gfCNCPoint5[23995] = {X 332.1055, Y 45.0114, Z -7.1667, A 0.000, B 0.000, C 0.000 }
gfCNCPoint5[23996] = {X 330.6899, Y 43.7933, Z -7.1667, A 0.000, B 0.000, C 0.000 }
gfCNCPoint5[23997] = {X 329.7573, Y 43.7998, Z -7.1667, A 0.000, B 0.000, C 0.000 }
gfCNCPoint5[23998] = {X 328.8457, Y 43.6022, Z -7.1667, A 0.000, B 0.000, C 0.000 }
gfCNCPoint5[23999] = {X 327.9994, Y 43.2101, Z -7.1667, A 0.000, B 0.000, C 0.000 }
gfCNCPoint5[24000] = {X 327.2594, Y 42.6425, Z -7.1667, A 0.000, B 0.000, C 0.000 }
gfCNCPoint5[24001] = {X 326.6366, Y 42.0352, Z -7.1667, A 0.000, B 0.000, C 0.000 }
gfCNCPoint5[24002] = {X 326.0198, Y 41.2760, Z -7.1667, A 0.000, B 0.000, C 0.000 }
gfCNCPoint5[24003] = {X 325.5934, Y 40.3956, Z -7.1667, A 0.000, B 0.000, C 0.000 }
gfCNCPoint5[24004] = {X 325.3802, Y 39.4410, Z -7.1667, A 0.000, B 0.000, C 0.000 }
gfCNCPoint5[24005] = {X 325.3913, Y 38.4628, Z -7.1667, A 0.000, B 0.000, C 0.000 }
gfCNCPoint5[24006] = {X 325.6264, Y 37.5133, Z -7.1667, A 0.000, B 0.000, C 0.000 }
gfCNCPoint5[24007] = {X 326.0727, Y 36.6429, Z -7.1667, A 0.000, B 0.000, C 0.000 }
gfCNCPoint5[24008] = {X 330.3061, Y 30.3131, Z -7.1667, A 0.000, B 0.000, C 0.000 }
gfCNCPoint5[24009] = {X 330.8964, Y 29.6095, Z -7.1667, A 0.000, B 0.000, C 0.000 }
gfCNCPoint5[24010] = {X 331.6243, Y 29.0495, Z -7.1667, A 0.000, B 0.000, C 0.000 }
gfCNCPoint5[24011] = {X 332.4558, Y 28.6593, Z -7.1667, A 0.000, B 0.000, C 0.000 }
gfCNCPoint5[24012] = {X 333.3518, Y 28.4574, Z -7.1667, A 0.000, B 0.000, C 0.000 }
gfCNCPoint5[24013] = {X 334.2702, Y 28.4532, Z -7.1667, A 0.000, B 0.000, C 0.000 }
gfCNCPoint5[24014] = {X 335.1680, Y 28.6468, Z -7.1667, A 0.000, B 0.000, C 0.000 }
gfCNCPoint5[24015] = {X 336.0031, Y 29.0293, Z -7.1667, A 0.000, B 0.000, C 0.000 }
gfCNCPoint5[24016] = {X 336.7362, Y 29.5826, Z -7.1667, A 0.000, B 0.000, C 0.000 }
gfCNCPoint5[24017] = {X 337.3723, Y 30.1953, Z -7.1667, A 0.000, B 0.000, C 0.000 }
gfCNCPoint5[24018] = {X 338.0008, Y 30.9797, Z -7.1667, A 0.000, B 0.000, C 0.000 }
gfCNCPoint5[24019] = {X 338.4269, Y 31.8901, Z -7.1667, A 0.000, B 0.000, C 0.000 }
gfCNCPoint5[24020] = {X 338.6268, Y 32.8751, Z -7.1667, A 0.000, B 0.000, C 0.000 }
gfCNCPoint5[24021] = {X 338.5892, Y 33.8795, Z -7.1667, A 0.000, B 0.000, C 0.000 }
gfCNCPoint5[24022] = {X 339.4394, Y 34.6548, Z -7.1667, A 0.000, B 0.000, C 0.000 }
gfCNCPoint5[24023] = {X 340.5845, Y 35.5676, Z -7.1667, A 0.000, B 0.000, C 0.000 }
gfCNCPoint5[24024] = {X 341.8428, Y 36.3165, Z -7.1667, A 0.000, B 0.000, C 0.000 }
gfCNCPoint5[24025] = {X 343.1911, Y 36.8877, Z -7.1667, A 0.000, B 0.000, C 0.000 }
gfCNCPoint5[24026] = {X 344.6045, Y 37.2707, Z -7.1667, A 0.000, B 0.000, C 0.000 }
gfCNCPoint5[24027] = {X 346.0568, Y 37.4583, Z -7.1667, A 0.000, B 0.000, C 0.000 }
gfCNCPoint5[24028] = {X 347.5211, Y 37.4471, Z -7.1667, A 0.000, B 0.000, C 0.000 }
gfCNCPoint5[24029] = {X 348.6869, Y 37.3101, Z -7.1667, A 0.000, B 0.000, C 0.000 }
gfCNCPoint5[24030] = {X 349.8249, Y 37.0222, Z -7.1667, A 0.000, B 0.000, C 0.000 }
gfCNCPoint5[24031] = {X 350.9155, Y 36.5881, Z -7.1667, A 0.000, B 0.000, C 0.000 }
gfCNCPoint5[24032] = {X 351.9402, Y 36.0155, Z -7.1667, A 0.000, B 0.000, C 0.000 }
gfCNCPoint5[24033] = {X 352.8814, Y 35.3139, Z -7.1667, A 0.000, B 0.000, C 0.000 }
gfCNCPoint5[24034] = {X 354.0420, Y 34.1861, Z -7.1667, A 0.000, B 0.000, C 0.000 }
gfCNCPoint5[24035] = {X 355.0465, Y 32.9171, Z -7.1667, A 0.000, B 0.000, C 0.000 }
gfCNCPoint5[24036] = {X 355.8777, Y 31.5284, Z -7.1667, A 0.000, B 0.000, C 0.000 }
gfCNCPoint5[24037] = {X 356.5216, Y 30.0436, Z -7.1667, A 0.000, B 0.000, C 0.000 }
gfCNCPoint5[24038] = {X 356.9674, Y 28.4878, Z -7.1667, A 0.000, B 0.000, C 0.000 }
gfCNCPoint5[24039] = {X 357.2419, Y 26.7920, Z -7.1667, A 0.000, B 0.000, C 0.000 }
gfCNCPoint5[24040] = {X 357.3537, Y 25.0778, Z -7.1667, A 0.000, B 0.000, C 0.000 }
gfCNCPoint5[24041] = {X 357.3018, Y 23.3607, Z -7.1667, A 0.000, B 0.000, C 0.000 }
gfCNCPoint5[24042] = {X 357.0867, Y 21.6563, Z -7.1667, A 0.000, B 0.000, C 0.000 }
gfCNCPoint5[24043] = {X 356.7306, Y 20.1305, Z -7.1667, A 0.000, B 0.000, C 0.000 }
gfCNCPoint5[24044] = {X 356.1774, Y 18.6646, Z -7.1667, A 0.000, B 0.000, C 0.000 }
gfCNCPoint5[24045] = {X 355.4366, Y 17.2839, Z -7.1667, A 0.000, B 0.000, C 0.000 }
gfCNCPoint5[24046] = {X 354.5211, Y 16.0124, Z -7.1667, A 0.000, B 0.000, C 0.000 }
gfCNCPoint5[24047] = {X 353.6429, Y 15.0774, Z -7.1667, A 0.000, B 0.000, C 0.000 }
gfCNCPoint5[24048] = {X 352.6435, Y 14.2732, Z -7.1667, A 0.000, B 0.000, C 0.000 }
gfCNCPoint5[24049] = {X 351.5422, Y 13.6154, Z -7.1667, A 0.000, B 0.000, C 0.000 }
gfCNCPoint5[24050] = {X 350.3604, Y 13.1166, Z -7.1667, A 0.000, B 0.000, C 0.000 }
gfCNCPoint5[24051] = {X 349.1209, Y 12.7865, Z -7.1667, A 0.000, B 0.000, C 0.000 }
gfCNCPoint5[24052] = {X 347.3426, Y 12.5648, Z -7.1667, A 0.000, B 0.000, C 0.000 }
gfCNCPoint5[24053] = {X 345.5506, Y 12.5817, Z -7.1667, A 0.000, B 0.000, C 0.000 }
gfCNCPoint5[24054] = {X 343.7768, Y 12.8368, Z -7.1667, A 0.000, B 0.000, C 0.000 }
gfCNCPoint5[24055] = {X 342.0527, Y 13.3256, Z -7.1667, A 0.000, B 0.000, C 0.000 }
gfCNCPoint5[24056] = {X 340.4090, Y 14.0394, Z -7.1667, A 0.000, B 0.000, C 0.000 }
gfCNCPoint5[24057] = {X 338.8748, Y 14.9655, Z -7.1667, A 0.000, B 0.000, C 0.000 }
gfCNCPoint5[24058] = {X 338.8440, Y 15.8037, Z -7.1667, A 0.000, B 0.000, C 0.000 }
gfCNCPoint5[24059] = {X 338.6487, Y 16.6194, Z -7.1667, A 0.000, B 0.000, C 0.000 }
gfCNCPoint5[24060] = {X 338.2968, Y 17.3808, Z -7.1667, A 0.000, B 0.000, C 0.000 }
gfCNCPoint5[24061] = {X 337.8018, Y 18.0579, Z -7.1667, A 0.000, B 0.000, C 0.000 }
gfCNCPoint5[24062] = {X 337.1832, Y 18.6244, Z -7.1667, A 0.000, B 0.000, C 0.000 }
gfCNCPoint5[24063] = {X 336.4675, Y 19.1512, Z -7.1667, A 0.000, B 0.000, C 0.000 }
gfCNCPoint5[24064] = {X 335.6668, Y 19.6018, Z -7.1667, A 0.000, B 0.000, C 0.000 }
gfCNCPoint5[24065] = {X 334.7878, Y 19.8694, Z -7.1667, A 0.000, B 0.000, C 0.000 }
gfCNCPoint5[24066] = {X 333.8718, Y 19.9414, Z -7.1667, A 0.000, B 0.000, C 0.000 }
gfCNCPoint5[24067] = {X 332.9618, Y 19.8143, Z -7.1667, A 0.000, B 0.000, C 0.000 }
gfCNCPoint5[24068] = {X 332.1006, Y 19.4942, Z -7.1667, A 0.000, B 0.000, C 0.000 }
gfCNCPoint5[24069] = {X 331.3285, Y 18.9960, Z -7.1667, A 0.000, B 0.000, C 0.000 }
gfCNCPoint5[24070] = {X 330.6819, Y 18.3433, Z -7.1667, A 0.000, B 0.000, C 0.000 }
gfCNCPoint5[24071] = {X 330.1911, Y 17.5665, Z -7.1667, A 0.000, B 0.000, C 0.000 }
gfCNCPoint5[24072] = {X 326.6662, Y 10.3152, Z -7.1667, A 0.000, B 0.000, C 0.000 }
gfCNCPoint5[24073] = {X 326.3374, Y 9.3676, Z -7.1667, A 0.000, B 0.000, C 0.000 }
gfCNCPoint5[24074] = {X 326.2405, Y 8.3693, Z -7.1667, A 0.000, B 0.000, C 0.000 }
gfCNCPoint5[24075] = {X 326.3807, Y 7.3762, Z -7.1667, A 0.000, B 0.000, C 0.000 }
gfCNCPoint5[24076] = {X 326.7504, Y 6.4438, Z -7.1667, A 0.000, B 0.000, C 0.000 }
gfCNCPoint5[24077] = {X 327.3287, Y 5.6243, Z -7.1667, A 0.000, B 0.000, C 0.000 }
gfCNCPoint5[24078] = {X 328.0833, Y 4.9636, Z -7.1667, A 0.000, B 0.000, C 0.000 }
gfCNCPoint5[24079] = {X 328.7533, Y 4.5047, Z -7.1667, A 0.000, B 0.000, C 0.000 }
gfCNCPoint5[24080] = {X 329.6259, Y 4.0538, Z -7.1667, A 0.000, B 0.000, C 0.000 }
gfCNCPoint5[24081] = {X 330.5788, Y 3.8157, Z -7.1667, A 0.000, B 0.000, C 0.000 }
gfCNCPoint5[24082] = {X 331.5610, Y 3.8033, Z -7.1667, A 0.000, B 0.000, C 0.000 }
gfCNCPoint5[24083] = {X 332.5196, Y 4.0172, Z -7.1667, A 0.000, B 0.000, C 0.000 }
gfCNCPoint5[24084] = {X 334.1874, Y 3.0908, Z -7.1667, A 0.000, B 0.000, C 0.000 }
gfCNCPoint5[24085] = {X 335.9135, Y 2.2781, Z -7.1667, A 0.000, B 0.000, C 0.000 }
gfCNCPoint5[24086] = {X 338.0088, Y 1.4619, Z -7.1667, A 0.000, B 0.000, C 0.000 }
gfCNCPoint5[24087] = {X 340.1662, Y 0.8282, Z -7.1667, A 0.000, B 0.000, C 0.000 }
gfCNCPoint5[24088] = {X 342.3700, Y 0.3814, Z -7.1667, A 0.000, B 0.000, C 0.000 }
gfCNCPoint5[24089] = {X 344.6039, Y 0.1250, Z -7.1667, A 0.000, B 0.000, C 0.000 }
gfCNCPoint5[24090] = {X 346.8516, Y 0.0608, Z -7.1667, A 0.000, B 0.000, C 0.000 }
gfCNCPoint5[24091] = {X 349.0965, Y 0.1893, Z -7.1667, A 0.000, B 0.000, C 0.000 }
gfCNCPoint5[24092] = {X 351.3222, Y 0.5096, Z -7.1667, A 0.000, B 0.000, C 0.000 }
gfCNCPoint5[24093] = {X 351.5893, Y 0.5597, Z -7.1667, A 0.000, B 0.000, C 0.000 }
gfCNCPoint5[24094] = {X 352.3279, Y -3.3715, Z -7.1667, A 0.000, B 0.000, C 0.000 }
gfCNCPoint5[24095] = {X 351.5745, Y 0.6384, Z -7.1667, A 0.000, B 0.000, C 0.000 }
gfCNCPoint5[24096] = {X 351.8406, Y 0.6884, Z -7.1667, A 0.000, B 0.000, C 0.000 }
gfCNCPoint5[24097] = {X 353.9459, Y 1.2276, Z -7.1667, A 0.000, B 0.000, C 0.000 }
gfCNCPoint5[24098] = {X 355.9837, Y 1.9829, Z -7.1667, A 0.000, B 0.000, C 0.000 }
gfCNCPoint5[24099] = {X 357.9319, Y 2.9460, Z -7.1667, A 0.000, B 0.000, C 0.000 }
gfCNCPoint5[24100] = {X 359.7693, Y 4.1066, Z -7.1667, A 0.000, B 0.000, C 0.000 }
gfCNCPoint5[24101] = {X 361.4761, Y 5.4520, Z -7.1667, A 0.000, B 0.000, C 0.000 }
gfCNCPoint5[24102] = {X 363.0336, Y 6.9676, Z -7.1667, A 0.000, B 0.000, C 0.000 }
gfCNCPoint5[24103] = {X 364.5697, Y 8.8254, Z -7.1667, A 0.000, B 0.000, C 0.000 }
gfCNCPoint5[24104] = {X 365.9174, Y 10.8241, Z -7.1667, A 0.000, B 0.000, C 0.000 }
gfCNCPoint5[24105] = {X 367.0637, Y 12.9447, Z -7.1667, A 0.000, B 0.000, C 0.000 }
gfCNCPoint5[24106] = {X 367.9979, Y 15.1669, Z -7.1667, A 0.000, B 0.000, C 0.000 }
gfCNCPoint5[24107] = {X 368.7109, Y 17.4697, Z -7.1667, A 0.000, B 0.000, C 0.000 }
gfCNCPoint5[24108] = {X 369.1905, Y 19.7506, Z -7.1667, A 0.000, B 0.000, C 0.000 }
gfCNCPoint5[24109] = {X 369.4997, Y 22.0608, Z -7.1667, A 0.000, B 0.000, C 0.000 }
gfCNCPoint5[24110] = {X 369.6369, Y 24.3876, Z -7.1667, A 0.000, B 0.000, C 0.000 }
gfCNCPoint5[24111] = {X 369.6012, Y 26.7182, Z -7.1667, A 0.000, B 0.000, C 0.000 }
gfCNCPoint5[24112] = {X 369.3929, Y 29.0396, Z -7.1667, A 0.000, B 0.000, C 0.000 }
gfCNCPoint5[24113] = {X 369.0132, Y 31.3393, Z -7.1667, A 0.000, B 0.000, C 0.000 }
gfCNCPoint5[24114] = {X 368.4925, Y 33.4300, Z -7.1667, A 0.000, B 0.000, C 0.000 }
gfCNCPoint5[24115] = {X 367.7892, Y 35.4666, Z -7.1667, A 0.000, B 0.000, C 0.000 }
gfCNCPoint5[24116] = {X 366.9088, Y 37.4330, Z -7.1667, A 0.000, B 0.000, C 0.000 }
gfCNCPoint5[24117] = {X 365.8582, Y 39.3141, Z -7.1667, A 0.000, B 0.000, C 0.000 }
gfCNCPoint5[24118] = {X 364.6455, Y 41.0950, Z -7.1667, A 0.000, B 0.000, C 0.000 }
gfCNCPoint5[24119] = {X 364.5295, Y 41.2537, Z -7.1667, A 0.000, B 0.000, C 0.000 }
gfCNCPoint5[24120] = {X 363.1395, Y 42.9180, Z -7.1667, A 0.000, B 0.000, C 0.000 }
gfCNCPoint5[24121] = {X 361.5913, Y 44.4361, Z -7.1667, A 0.000, B 0.000, C 0.000 }
gfCNCPoint5[24122] = {X 359.9001, Y 45.7931, Z -7.1667, A 0.000, B 0.000, C 0.000 }
gfCNCPoint5[24123] = {X 358.0826, Y 46.9756, Z -7.1667, A 0.000, B 0.000, C 0.000 }
gfCNCPoint5[24124] = {X 356.1567, Y 47.9719, Z -7.1667, A 0.000, B 0.000, C 0.000 }
gfCNCPoint5[24125] = {X 353.9741, Y 48.7864, Z -7.1667, A 0.000, B 0.000, C 0.000 }
gfCNCPoint5[24126] = {X 351.7199, Y 49.3746, Z -7.1667, A 0.000, B 0.000, C 0.000 }
gfCNCPoint5[24127] = {X 349.4176, Y 49.7303, Z -7.1667, A 0.000, B 0.000, C 0.000 }
gfCNCPoint5[24128] = {X 347.0911, Y 49.8499, Z -7.1667, A 0.000, B 0.000, C 0.000 }
gfCNCPoint5[24129] = {X 345.0383, Y 49.8155, Z -7.1667, A 0.000, B 0.000, C 0.000 }
gfCNCPoint5[24130] = {X 342.9962, Y 49.6031, Z -7.1667, A 0.000, B 0.000, C 0.000 }
gfCNCPoint5[24131] = {X 340.9803, Y 49.2144, Z -7.1667, A 0.000, B 0.000, C 0.000 }
gfCNCPoint5[24132] = {X 339.0056, Y 48.6524, Z -7.1667, A 0.000, B 0.000, C 0.000 }
gfCNCPoint5[24133] = {X 337.0872, Y 47.9211, Z -7.1667, A 0.000, B 0.000, C 0.000 }
gfCNCPoint5[24134] = {X 335.2394, Y 47.0263, Z -7.1667, A 0.000, B 0.000, C 0.000 }
gfCNCPoint5[24135] = {X 333.6461, Y 46.0410, Z -7.1667, A 0.000, B 0.000, C 0.000 }
gfCNCPoint5[24136] = {X 332.1356, Y 44.9331, Z -7.1667, A 0.000, B 0.000, C 0.000 }
gfCNCPoint5[24137] = {X 330.7172, Y 43.7094, Z -7.1667, A 0.000, B 0.000, C 0.000 }
gfCNCPoint5[24138] = {X 329.7931, Y 43.7230, Z -7.1667, A 0.000, B 0.000, C 0.000 }
gfCNCPoint5[24139] = {X 328.8887, Y 43.5322, Z -7.1667, A 0.000, B 0.000, C 0.000 }
gfCNCPoint5[24140] = {X 328.0488, Y 43.1465, Z -7.1667, A 0.000, B 0.000, C 0.000 }
gfCNCPoint5[24141] = {X 327.3148, Y 42.5847, Z -7.1667, A 0.000, B 0.000, C 0.000 }
gfCNCPoint5[24142] = {X 326.6925, Y 41.9780, Z -7.1667, A 0.000, B 0.000, C 0.000 }
gfCNCPoint5[24143] = {X 326.0873, Y 41.2331, Z -7.1667, A 0.000, B 0.000, C 0.000 }
gfCNCPoint5[24144] = {X 325.6690, Y 40.3693, Z -7.1667, A 0.000, B 0.000, C 0.000 }
gfCNCPoint5[24145] = {X 325.4597, Y 39.4326, Z -7.1667, A 0.000, B 0.000, C 0.000 }
gfCNCPoint5[24146] = {X 325.4707, Y 38.4730, Z -7.1667, A 0.000, B 0.000, C 0.000 }
gfCNCPoint5[24147] = {X 325.7013, Y 37.5413, Z -7.1667, A 0.000, B 0.000, C 0.000 }
gfCNCPoint5[24148] = {X 326.1392, Y 36.6874, Z -7.1667, A 0.000, B 0.000, C 0.000 }
gfCNCPoint5[24149] = {X 330.3726, Y 30.3576, Z -7.1667, A 0.000, B 0.000, C 0.000 }
gfCNCPoint5[24150] = {X 330.9517, Y 29.6673, Z -7.1667, A 0.000, B 0.000, C 0.000 }
gfCNCPoint5[24151] = {X 331.6658, Y 29.1178, Z -7.1667, A 0.000, B 0.000, C 0.000 }
gfCNCPoint5[24152] = {X 332.4816, Y 28.7351, Z -7.1667, A 0.000, B 0.000, C 0.000 }
gfCNCPoint5[24153] = {X 333.3606, Y 28.5369, Z -7.1667, A 0.000, B 0.000, C 0.000 }
gfCNCPoint5[24154] = {X 334.2616, Y 28.5327, Z -7.1667, A 0.000, B 0.000, C 0.000 }
gfCNCPoint5[24155] = {X 335.1425, Y 28.7227, Z -7.1667, A 0.000, B 0.000, C 0.000 }
gfCNCPoint5[24156] = {X 335.9617, Y 29.0978, Z -7.1667, A 0.000, B 0.000, C 0.000 }
gfCNCPoint5[24157] = {X 336.6810, Y 29.6405, Z -7.1667, A 0.000, B 0.000, C 0.000 }
gfCNCPoint5[24158] = {X 337.3163, Y 30.2523, Z -7.1667, A 0.000, B 0.000, C 0.000 }
gfCNCPoint5[24159] = {X 337.8297, Y 30.8643, Z -7.1667, A 0.000, B 0.000, C 0.000 }
gfCNCPoint5[24160] = {X 338.2167, Y 31.5631, Z -7.1667, A 0.000, B 0.000, C 0.000 }
gfCNCPoint5[24161] = {X 338.4630, Y 32.3230, Z -7.1667, A 0.000, B 0.000, C 0.000 }
gfCNCPoint5[24162] = {X 338.5595, Y 33.1159, Z -7.1667, A 0.000, B 0.000, C 0.000 }
gfCNCPoint5[24163] = {X 338.5027, Y 33.9127, Z -7.1667, A 0.000, B 0.000, C 0.000 }
gfCNCPoint5[24164] = {X 338.5556, Y 33.9552, Z -7.1667, A 0.000, B 0.000, C 0.000 }
gfCNCPoint5[24165] = {X 339.3854, Y 34.7138, Z -7.1667, A 0.000, B 0.000, C 0.000 }
gfCNCPoint5[24166] = {X 340.5388, Y 35.6333, Z -7.1667, A 0.000, B 0.000, C 0.000 }
gfCNCPoint5[24167] = {X 341.8064, Y 36.3877, Z -7.1667, A 0.000, B 0.000, C 0.000 }
gfCNCPoint5[24168] = {X 343.1645, Y 36.9632, Z -7.1667, A 0.000, B 0.000, C 0.000 }
gfCNCPoint5[24169] = {X 344.5883, Y 37.3490, Z -7.1667, A 0.000, B 0.000, C 0.000 }
gfCNCPoint5[24170] = {X 346.0511, Y 37.5381, Z -7.1667, A 0.000, B 0.000, C 0.000 }
gfCNCPoint5[24171] = {X 347.5262, Y 37.5269, Z -7.1667, A 0.000, B 0.000, C 0.000 }
gfCNCPoint5[24172] = {X 348.7022, Y 37.3887, Z -7.1667, A 0.000, B 0.000, C 0.000 }
gfCNCPoint5[24173] = {X 349.8501, Y 37.0981, Z -7.1667, A 0.000, B 0.000, C 0.000 }
gfCNCPoint5[24174] = {X 350.9503, Y 36.6602, Z -7.1667, A 0.000, B 0.000, C 0.000 }
gfCNCPoint5[24175] = {X 351.9839, Y 36.0825, Z -7.1667, A 0.000, B 0.000, C 0.000 }
gfCNCPoint5[24176] = {X 352.9333, Y 35.3748, Z -7.1667, A 0.000, B 0.000, C 0.000 }
gfCNCPoint5[24177] = {X 354.1014, Y 34.2396, Z -7.1667, A 0.000, B 0.000, C 0.000 }
gfCNCPoint5[24178] = {X 355.1123, Y 32.9624, Z -7.1667, A 0.000, B 0.000, C 0.000 }
gfCNCPoint5[24179] = {X 355.9489, Y 31.5648, Z -7.1667, A 0.000, B 0.000, C 0.000 }
gfCNCPoint5[24180] = {X 356.5970, Y 30.0704, Z -7.1667, A 0.000, B 0.000, C 0.000 }
gfCNCPoint5[24181] = {X 357.0456, Y 28.5046, Z -7.1667, A 0.000, B 0.000, C 0.000 }
gfCNCPoint5[24182] = {X 357.3213, Y 26.8012, Z -7.1667, A 0.000, B 0.000, C 0.000 }
gfCNCPoint5[24183] = {X 357.4336, Y 25.0793, Z -7.1667, A 0.000, B 0.000, C 0.000 }
gfCNCPoint5[24184] = {X 357.3815, Y 23.3545, Z -7.1667, A 0.000, B 0.000, C 0.000 }
gfCNCPoint5[24185] = {X 357.1655, Y 21.6425, Z -7.1667, A 0.000, B 0.000, C 0.000 }
gfCNCPoint5[24186] = {X 356.8069, Y 20.1067, Z -7.1667, A 0.000, B 0.000, C 0.000 }
gfCNCPoint5[24187] = {X 356.2500, Y 18.6311, Z -7.1667, A 0.000, B 0.000, C 0.000 }
gfCNCPoint5[24188] = {X 355.5043, Y 17.2414, Z -7.1667, A 0.000, B 0.000, C 0.000 }
gfCNCPoint5[24189] = {X 354.5828, Y 15.9615, Z -7.1667, A 0.000, B 0.000, C 0.000 }
gfCNCPoint5[24190] = {X 353.6970, Y 15.0185, Z -7.1667, A 0.000, B 0.000, C 0.000 }
gfCNCPoint5[24191] = {X 352.6890, Y 14.2074, Z -7.1667, A 0.000, B 0.000, C 0.000 }
gfCNCPoint5[24192] = {X 351.5782, Y 13.5440, Z -7.1667, A 0.000, B 0.000, C 0.000 }
gfCNCPoint5[24193] = {X 350.3863, Y 13.0409, Z -7.1667, A 0.000, B 0.000, C 0.000 }
gfCNCPoint5[24194] = {X 349.1360, Y 12.7080, Z -7.1667, A 0.000, B 0.000, C 0.000 }
gfCNCPoint5[24195] = {X 347.5979, Y 12.5017, Z -7.1667, A 0.000, B 0.000, C 0.000 }
gfCNCPoint5[24196] = {X 346.0462, Y 12.4730, Z -7.1667, A 0.000, B 0.000, C 0.000 }
gfCNCPoint5[24197] = {X 344.5014, Y 12.6224, Z -7.1667, A 0.000, B 0.000, C 0.000 }
gfCNCPoint5[24198] = {X 342.9840, Y 12.9477, Z -7.1667, A 0.000, B 0.000, C 0.000 }
gfCNCPoint5[24199] = {X 341.5138, Y 13.4449, Z -7.1667, A 0.000, B 0.000, C 0.000 }
gfCNCPoint5[24200] = {X 340.1103, Y 14.1071, Z -7.1667, A 0.000, B 0.000, C 0.000 }
gfCNCPoint5[24201] = {X 338.7919, Y 14.9259, Z -7.1667, A 0.000, B 0.000, C 0.000 }
gfCNCPoint5[24202] = {X 338.7694, Y 15.7574, Z -7.1667, A 0.000, B 0.000, C 0.000 }
gfCNCPoint5[24203] = {X 338.5819, Y 16.5679, Z -7.1667, A 0.000, B 0.000, C 0.000 }
gfCNCPoint5[24204] = {X 338.2369, Y 17.3248, Z -7.1667, A 0.000, B 0.000, C 0.000 }
gfCNCPoint5[24205] = {X 337.7482, Y 17.9979, Z -7.1667, A 0.000, B 0.000, C 0.000 }
gfCNCPoint5[24206] = {X 337.1353, Y 18.5604, Z -7.1667, A 0.000, B 0.000, C 0.000 }
gfCNCPoint5[24207] = {X 336.4209, Y 19.0861, Z -7.1667, A 0.000, B 0.000, C 0.000 }
gfCNCPoint5[24208] = {X 335.6353, Y 19.5283, Z -7.1667, A 0.000, B 0.000, C 0.000 }
gfCNCPoint5[24209] = {X 334.7729, Y 19.7908, Z -7.1667, A 0.000, B 0.000, C 0.000 }
gfCNCPoint5[24210] = {X 333.8742, Y 19.8614, Z -7.1667, A 0.000, B 0.000, C 0.000 }
gfCNCPoint5[24211] = {X 332.9814, Y 19.7367, Z -7.1667, A 0.000, B 0.000, C 0.000 }
gfCNCPoint5[24212] = {X 332.1364, Y 19.4226, Z -7.1667, A 0.000, B 0.000, C 0.000 }
gfCNCPoint5[24213] = {X 331.3789, Y 18.9339, Z -7.1667, A 0.000, B 0.000, C 0.000 }
gfCNCPoint5[24214] = {X 330.7445, Y 18.2934, Z -7.1667, A 0.000, B 0.000, C 0.000 }
gfCNCPoint5[24215] = {X 330.2630, Y 17.5314, Z -7.1667, A 0.000, B 0.000, C 0.000 }
gfCNCPoint5[24216] = {X 326.7381, Y 10.2803, Z -7.1667, A 0.000, B 0.000, C 0.000 }
gfCNCPoint5[24217] = {X 326.4156, Y 9.3505, Z -7.1667, A 0.000, B 0.000, C 0.000 }
gfCNCPoint5[24218] = {X 326.3205, Y 8.3711, Z -7.1667, A 0.000, B 0.000, C 0.000 }
gfCNCPoint5[24219] = {X 326.4581, Y 7.3967, Z -7.1667, A 0.000, B 0.000, C 0.000 }
gfCNCPoint5[24220] = {X 326.8207, Y 6.4819, Z -7.1667, A 0.000, B 0.000, C 0.000 }
gfCNCPoint5[24221] = {X 327.3881, Y 5.6778, Z -7.1667, A 0.000, B 0.000, C 0.000 }
gfCNCPoint5[24222] = {X 328.1285, Y 5.0296, Z -7.1667, A 0.000, B 0.000, C 0.000 }
gfCNCPoint5[24223] = {X 328.7983, Y 4.5709, Z -7.1667, A 0.000, B 0.000, C 0.000 }
gfCNCPoint5[24224] = {X 329.6631, Y 4.1253, Z -7.1667, A 0.000, B 0.000, C 0.000 }
gfCNCPoint5[24225] = {X 330.6078, Y 3.8927, Z -7.1667, A 0.000, B 0.000, C 0.000 }
gfCNCPoint5[24226] = {X 331.5806, Y 3.8859, Z -7.1667, A 0.000, B 0.000, C 0.000 }
gfCNCPoint5[24227] = {X 332.5285, Y 4.1052, Z -7.1667, A 0.000, B 0.000, C 0.000 }
gfCNCPoint5[24228] = {X 334.2073, Y 3.1705, Z -7.1667, A 0.000, B 0.000, C 0.000 }
gfCNCPoint5[24229] = {X 335.9455, Y 2.3514, Z -7.1667, A 0.000, B 0.000, C 0.000 }
gfCNCPoint5[24230] = {X 338.0344, Y 1.5377, Z -7.1667, A 0.000, B 0.000, C 0.000 }
gfCNCPoint5[24231] = {X 340.1853, Y 0.9059, Z -7.1667, A 0.000, B 0.000, C 0.000 }
gfCNCPoint5[24232] = {X 342.3823, Y 0.4605, Z -7.1667, A 0.000, B 0.000, C 0.000 }
gfCNCPoint5[24233] = {X 344.6095, Y 0.2048, Z -7.1667, A 0.000, B 0.000, C 0.000 }
gfCNCPoint5[24234] = {X 346.8504, Y 0.1408, Z -7.1667, A 0.000, B 0.000, C 0.000 }
gfCNCPoint5[24235] = {X 349.0885, Y 0.2689, Z -7.1667, A 0.000, B 0.000, C 0.000 }
gfCNCPoint5[24236] = {X 351.3074, Y 0.5882, Z -7.1667, A 0.000, B 0.000, C 0.000 }
gfCNCPoint5[24237] = {X 351.5745, Y 0.6384, Z -7.1667, A 0.000, B 0.000, C 0.000 }
gfCNCPoint5[24238] = {X 352.3131, Y -3.2928, Z -7.1667, A 0.000, B 0.000, C 0.000 }
gfCNCPoint5[24239] = {X 351.5598, Y 0.7170, Z -7.1667, A 0.000, B 0.000, C 0.000 }
gfCNCPoint5[24240] = {X 351.8254, Y 0.7669, Z -7.1667, A 0.000, B 0.000, C 0.000 }
gfCNCPoint5[24241] = {X 353.9225, Y 1.3041, Z -7.1667, A 0.000, B 0.000, C 0.000 }
gfCNCPoint5[24242] = {X 355.9524, Y 2.0565, Z -7.1667, A 0.000, B 0.000, C 0.000 }
gfCNCPoint5[24243] = {X 357.8930, Y 3.0159, Z -7.1667, A 0.000, B 0.000, C 0.000 }
gfCNCPoint5[24244] = {X 359.7233, Y 4.1720, Z -7.1667, A 0.000, B 0.000, C 0.000 }
gfCNCPoint5[24245] = {X 361.4234, Y 5.5122, Z -7.1667, A 0.000, B 0.000, C 0.000 }
gfCNCPoint5[24246] = {X 362.9749, Y 7.0219, Z -7.1667, A 0.000, B 0.000, C 0.000 }
gfCNCPoint5[24247] = {X 364.5059, Y 8.8737, Z -7.1667, A 0.000, B 0.000, C 0.000 }
gfCNCPoint5[24248] = {X 365.8491, Y 10.8658, Z -7.1667, A 0.000, B 0.000, C 0.000 }
gfCNCPoint5[24249] = {X 366.9917, Y 12.9795, Z -7.1667, A 0.000, B 0.000, C 0.000 }
gfCNCPoint5[24250] = {X 367.9227, Y 15.1944, Z -7.1667, A 0.000, B 0.000, C 0.000 }
gfCNCPoint5[24251] = {X 368.6334, Y 17.4896, Z -7.1667, A 0.000, B 0.000, C 0.000 }
gfCNCPoint5[24252] = {X 369.1117, Y 19.7646, Z -7.1667, A 0.000, B 0.000, C 0.000 }
gfCNCPoint5[24253] = {X 369.4201, Y 22.0689, Z -7.1667, A 0.000, B 0.000, C 0.000 }
gfCNCPoint5[24254] = {X 369.5569, Y 24.3896, Z -7.1667, A 0.000, B 0.000, C 0.000 }
gfCNCPoint5[24255] = {X 369.5213, Y 26.7142, Z -7.1667, A 0.000, B 0.000, C 0.000 }
gfCNCPoint5[24256] = {X 369.3136, Y 29.0296, Z -7.1667, A 0.000, B 0.000, C 0.000 }
gfCNCPoint5[24257] = {X 368.9348, Y 31.3234, Z -7.1667, A 0.000, B 0.000, C 0.000 }
gfCNCPoint5[24258] = {X 368.4158, Y 33.4073, Z -7.1667, A 0.000, B 0.000, C 0.000 }
gfCNCPoint5[24259] = {X 367.7147, Y 35.4372, Z -7.1667, A 0.000, B 0.000, C 0.000 }
gfCNCPoint5[24260] = {X 366.8372, Y 37.3974, Z -7.1667, A 0.000, B 0.000, C 0.000 }
gfCNCPoint5[24261] = {X 365.7899, Y 39.2723, Z -7.1667, A 0.000, B 0.000, C 0.000 }
gfCNCPoint5[24262] = {X 364.5812, Y 41.0474, Z -7.1667, A 0.000, B 0.000, C 0.000 }
gfCNCPoint5[24263] = {X 364.4652, Y 41.2060, Z -7.1667, A 0.000, B 0.000, C 0.000 }
gfCNCPoint5[24264] = {X 363.0805, Y 42.8639, Z -7.1667, A 0.000, B 0.000, C 0.000 }
gfCNCPoint5[24265] = {X 361.5382, Y 44.3763, Z -7.1667, A 0.000, B 0.000, C 0.000 }
gfCNCPoint5[24266] = {X 359.8534, Y 45.7282, Z -7.1667, A 0.000, B 0.000, C 0.000 }
gfCNCPoint5[24267] = {X 358.0428, Y 46.9062, Z -7.1667, A 0.000, B 0.000, C 0.000 }
gfCNCPoint5[24268] = {X 356.1242, Y 47.8988, Z -7.1667, A 0.000, B 0.000, C 0.000 }
gfCNCPoint5[24269] = {X 353.9491, Y 48.7104, Z -7.1667, A 0.000, B 0.000, C 0.000 }
gfCNCPoint5[24270] = {X 351.7028, Y 49.2964, Z -7.1667, A 0.000, B 0.000, C 0.000 }
gfCNCPoint5[24271] = {X 349.4085, Y 49.6508, Z -7.1667, A 0.000, B 0.000, C 0.000 }
gfCNCPoint5[24272] = {X 347.0900, Y 49.7699, Z -7.1667, A 0.000, B 0.000, C 0.000 }
gfCNCPoint5[24273] = {X 345.0441, Y 49.7357, Z -7.1667, A 0.000, B 0.000, C 0.000 }
gfCNCPoint5[24274] = {X 343.0089, Y 49.5241, Z -7.1667, A 0.000, B 0.000, C 0.000 }
gfCNCPoint5[24275] = {X 340.9997, Y 49.1368, Z -7.1667, A 0.000, B 0.000, C 0.000 }
gfCNCPoint5[24276] = {X 339.0317, Y 48.5767, Z -7.1667, A 0.000, B 0.000, C 0.000 }
gfCNCPoint5[24277] = {X 337.1196, Y 47.8480, Z -7.1667, A 0.000, B 0.000, C 0.000 }
gfCNCPoint5[24278] = {X 335.2780, Y 46.9562, Z -7.1667, A 0.000, B 0.000, C 0.000 }
gfCNCPoint5[24279] = {X 333.6800, Y 45.9674, Z -7.1667, A 0.000, B 0.000, C 0.000 }
gfCNCPoint5[24280] = {X 332.1655, Y 44.8547, Z -7.1667, A 0.000, B 0.000, C 0.000 }
gfCNCPoint5[24281] = {X 330.7443, Y 43.6252, Z -7.1667, A 0.000, B 0.000, C 0.000 }
gfCNCPoint5[24282] = {X 329.8287, Y 43.6460, Z -7.1667, A 0.000, B 0.000, C 0.000 }
gfCNCPoint5[24283] = {X 328.9316, Y 43.4621, Z -7.1667, A 0.000, B 0.000, C 0.000 }
gfCNCPoint5[24284] = {X 328.0980, Y 43.0827, Z -7.1667, A 0.000, B 0.000, C 0.000 }
gfCNCPoint5[24285] = {X 327.3701, Y 42.5270, Z -7.1667, A 0.000, B 0.000, C 0.000 }
gfCNCPoint5[24286] = {X 326.7483, Y 41.9207, Z -7.1667, A 0.000, B 0.000, C 0.000 }
gfCNCPoint5[24287] = {X 326.1548, Y 41.1901, Z -7.1667, A 0.000, B 0.000, C 0.000 }
gfCNCPoint5[24288] = {X 325.7445, Y 40.3430, Z -7.1667, A 0.000, B 0.000, C 0.000 }
gfCNCPoint5[24289] = {X 325.5393, Y 39.4243, Z -7.1667, A 0.000, B 0.000, C 0.000 }
gfCNCPoint5[24290] = {X 325.5500, Y 38.4831, Z -7.1667, A 0.000, B 0.000, C 0.000 }
gfCNCPoint5[24291] = {X 325.7762, Y 37.5694, Z -7.1667, A 0.000, B 0.000, C 0.000 }
gfCNCPoint5[24292] = {X 326.2057, Y 36.7318, Z -7.1667, A 0.000, B 0.000, C 0.000 }
gfCNCPoint5[24293] = {X 330.4391, Y 30.4021, Z -7.1667, A 0.000, B 0.000, C 0.000 }
gfCNCPoint5[24294] = {X 331.0070, Y 29.7251, Z -7.1667, A 0.000, B 0.000, C 0.000 }
gfCNCPoint5[24295] = {X 331.7074, Y 29.1862, Z -7.1667, A 0.000, B 0.000, C 0.000 }
gfCNCPoint5[24296] = {X 332.5074, Y 28.8108, Z -7.1667, A 0.000, B 0.000, C 0.000 }
gfCNCPoint5[24297] = {X 333.3694, Y 28.6165, Z -7.1667, A 0.000, B 0.000, C 0.000 }
gfCNCPoint5[24298] = {X 334.2531, Y 28.6123, Z -7.1667, A 0.000, B 0.000, C 0.000 }
gfCNCPoint5[24299] = {X 335.1169, Y 28.7985, Z -7.1667, A 0.000, B 0.000, C 0.000 }
gfCNCPoint5[24300] = {X 335.9204, Y 29.1663, Z -7.1667, A 0.000, B 0.000, C 0.000 }
gfCNCPoint5[24301] = {X 336.6259, Y 29.6985, Z -7.1667, A 0.000, B 0.000, C 0.000 }
gfCNCPoint5[24302] = {X 337.2602, Y 30.3094, Z -7.1667, A 0.000, B 0.000, C 0.000 }
gfCNCPoint5[24303] = {X 337.8541, Y 31.0469, Z -7.1667, A 0.000, B 0.000, C 0.000 }
gfCNCPoint5[24304] = {X 338.2619, Y 31.9014, Z -7.1667, A 0.000, B 0.000, C 0.000 }
gfCNCPoint5[24305] = {X 338.4618, Y 32.8269, Z -7.1667, A 0.000, B 0.000, C 0.000 }
gfCNCPoint5[24306] = {X 338.4431, Y 33.7735, Z -7.1667, A 0.000, B 0.000, C 0.000 }
gfCNCPoint5[24307] = {X 338.4303, Y 33.8596, Z -7.1667, A 0.000, B 0.000, C 0.000 }
gfCNCPoint5[24308] = {X 338.4158, Y 33.9455, Z -7.1667, A 0.000, B 0.000, C 0.000 }
gfCNCPoint5[24309] = {X 338.5035, Y 34.0159, Z -7.1667, A 0.000, B 0.000, C 0.000 }
gfCNCPoint5[24310] = {X 339.3314, Y 34.7729, Z -7.1667, A 0.000, B 0.000, C 0.000 }
gfCNCPoint5[24311] = {X 340.4932, Y 35.6990, Z -7.1667, A 0.000, B 0.000, C 0.000 }
gfCNCPoint5[24312] = {X 341.7699, Y 36.4589, Z -7.1667, A 0.000, B 0.000, C 0.000 }
gfCNCPoint5[24313] = {X 343.1380, Y 37.0386, Z -7.1667, A 0.000, B 0.000, C 0.000 }
gfCNCPoint5[24314] = {X 344.5720, Y 37.4273, Z -7.1667, A 0.000, B 0.000, C 0.000 }
gfCNCPoint5[24315] = {X 346.0455, Y 37.6179, Z -7.1667, A 0.000, B 0.000, C 0.000 }
gfCNCPoint5[24316] = {X 347.5312, Y 37.6068, Z -7.1667, A 0.000, B 0.000, C 0.000 }
gfCNCPoint5[24317] = {X 348.7175, Y 37.4672, Z -7.1667, A 0.000, B 0.000, C 0.000 }
gfCNCPoint5[24318] = {X 349.8753, Y 37.1740, Z -7.1667, A 0.000, B 0.000, C 0.000 }
gfCNCPoint5[24319] = {X 350.9850, Y 36.7323, Z -7.1667, A 0.000, B 0.000, C 0.000 }
gfCNCPoint5[24320] = {X 352.0276, Y 36.1495, Z -7.1667, A 0.000, B 0.000, C 0.000 }
gfCNCPoint5[24321] = {X 352.9852, Y 35.4357, Z -7.1667, A 0.000, B 0.000, C 0.000 }
gfCNCPoint5[24322] = {X 354.1608, Y 34.2932, Z -7.1667, A 0.000, B 0.000, C 0.000 }
gfCNCPoint5[24323] = {X 355.1782, Y 33.0078, Z -7.1667, A 0.000, B 0.000, C 0.000 }
gfCNCPoint5[24324] = {X 356.0201, Y 31.6013, Z -7.1667, A 0.000, B 0.000, C 0.000 }
gfCNCPoint5[24325] = {X 356.6724, Y 30.0973, Z -7.1667, A 0.000, B 0.000, C 0.000 }
gfCNCPoint5[24326] = {X 357.1238, Y 28.5214, Z -7.1667, A 0.000, B 0.000, C 0.000 }
gfCNCPoint5[24327] = {X 357.4008, Y 26.8104, Z -7.1667, A 0.000, B 0.000, C 0.000 }
gfCNCPoint5[24328] = {X 357.5136, Y 25.0808, Z -7.1667, A 0.000, B 0.000, C 0.000 }
gfCNCPoint5[24329] = {X 357.4613, Y 23.3484, Z -7.1667, A 0.000, B 0.000, C 0.000 }
gfCNCPoint5[24330] = {X 357.2443, Y 21.6288, Z -7.1667, A 0.000, B 0.000, C 0.000 }
gfCNCPoint5[24331] = {X 356.8833, Y 20.0829, Z -7.1667, A 0.000, B 0.000, C 0.000 }
gfCNCPoint5[24332] = {X 356.3227, Y 18.5977, Z -7.1667, A 0.000, B 0.000, C 0.000 }
gfCNCPoint5[24333] = {X 355.5721, Y 17.1988, Z -7.1667, A 0.000, B 0.000, C 0.000 }
gfCNCPoint5[24334] = {X 354.6445, Y 15.9106, Z -7.1667, A 0.000, B 0.000, C 0.000 }
gfCNCPoint5[24335] = {X 353.7511, Y 14.9596, Z -7.1667, A 0.000, B 0.000, C 0.000 }
gfCNCPoint5[24336] = {X 352.7345, Y 14.1416, Z -7.1667, A 0.000, B 0.000, C 0.000 }
gfCNCPoint5[24337] = {X 351.6142, Y 13.4725, Z -7.1667, A 0.000, B 0.000, C 0.000 }
gfCNCPoint5[24338] = {X 350.4121, Y 12.9652, Z -7.1667, A 0.000, B 0.000, C 0.000 }
gfCNCPoint5[24339] = {X 349.1512, Y 12.6294, Z -7.1667, A 0.000, B 0.000, C 0.000 }
gfCNCPoint5[24340] = {X 347.5974, Y 12.4214, Z -7.1667, A 0.000, B 0.000, C 0.000 }
gfCNCPoint5[24341] = {X 346.0300, Y 12.3936, Z -7.1667, A 0.000, B 0.000, C 0.000 }
gfCNCPoint5[24342] = {X 344.4699, Y 12.5463, Z -7.1667, A 0.000, B 0.000, C 0.000 }
gfCNCPoint5[24343] = {X 342.9376, Y 12.8776, Z -7.1667, A 0.000, B 0.000, C 0.000 }
gfCNCPoint5[24344] = {X 341.4537, Y 13.3829, Z -7.1667, A 0.000, B 0.000, C 0.000 }
gfCNCPoint5[24345] = {X 340.0377, Y 14.0556, Z -7.1667, A 0.000, B 0.000, C 0.000 }
gfCNCPoint5[24346] = {X 338.7086, Y 14.8868, Z -7.1667, A 0.000, B 0.000, C 0.000 }
gfCNCPoint5[24347] = {X 338.6944, Y 15.7115, Z -7.1667, A 0.000, B 0.000, C 0.000 }
gfCNCPoint5[24348] = {X 338.5147, Y 16.5165, Z -7.1667, A 0.000, B 0.000, C 0.000 }
gfCNCPoint5[24349] = {X 338.1768, Y 17.2689, Z -7.1667, A 0.000, B 0.000, C 0.000 }
gfCNCPoint5[24350] = {X 337.6944, Y 17.9379, Z -7.1667, A 0.000, B 0.000, C 0.000 }
gfCNCPoint5[24351] = {X 337.0874, Y 18.4963, Z -7.1667, A 0.000, B 0.000, C 0.000 }
gfCNCPoint5[24352] = {X 336.3744, Y 19.0211, Z -7.1667, A 0.000, B 0.000, C 0.000 }
gfCNCPoint5[24353] = {X 335.6039, Y 19.4547, Z -7.1667, A 0.000, B 0.000, C 0.000 }
gfCNCPoint5[24354] = {X 334.7580, Y 19.7122, Z -7.1667, A 0.000, B 0.000, C 0.000 }
gfCNCPoint5[24355] = {X 333.8766, Y 19.7814, Z -7.1667, A 0.000, B 0.000, C 0.000 }
gfCNCPoint5[24356] = {X 333.0010, Y 19.6592, Z -7.1667, A 0.000, B 0.000, C 0.000 }
gfCNCPoint5[24357] = {X 332.1722, Y 19.3511, Z -7.1667, A 0.000, B 0.000, C 0.000 }
gfCNCPoint5[24358] = {X 331.4293, Y 18.8718, Z -7.1667, A 0.000, B 0.000, C 0.000 }
gfCNCPoint5[24359] = {X 330.8071, Y 18.2436, Z -7.1667, A 0.000, B 0.000, C 0.000 }
gfCNCPoint5[24360] = {X 330.3348, Y 17.4962, Z -7.1667, A 0.000, B 0.000, C 0.000 }
gfCNCPoint5[24361] = {X 326.8100, Y 10.2453, Z -7.1667, A 0.000, B 0.000, C 0.000 }
gfCNCPoint5[24362] = {X 326.4937, Y 9.3334, Z -7.1667, A 0.000, B 0.000, C 0.000 }
gfCNCPoint5[24363] = {X 326.4004, Y 8.3728, Z -7.1667, A 0.000, B 0.000, C 0.000 }
gfCNCPoint5[24364] = {X 326.5354, Y 7.4171, Z -7.1667, A 0.000, B 0.000, C 0.000 }
gfCNCPoint5[24365] = {X 326.8911, Y 6.5199, Z -7.1667, A 0.000, B 0.000, C 0.000 }
gfCNCPoint5[24366] = {X 327.4476, Y 5.7314, Z -7.1667, A 0.000, B 0.000, C 0.000 }
gfCNCPoint5[24367] = {X 328.1737, Y 5.0956, Z -7.1667, A 0.000, B 0.000, C 0.000 }
gfCNCPoint5[24368] = {X 328.8432, Y 4.6371, Z -7.1667, A 0.000, B 0.000, C 0.000 }
gfCNCPoint5[24369] = {X 329.7002, Y 4.1968, Z -7.1667, A 0.000, B 0.000, C 0.000 }
gfCNCPoint5[24370] = {X 330.6366, Y 3.9698, Z -7.1667, A 0.000, B 0.000, C 0.000 }
gfCNCPoint5[24371] = {X 331.6001, Y 3.9686, Z -7.1667, A 0.000, B 0.000, C 0.000 }
gfCNCPoint5[24372] = {X 332.5370, Y 4.1935, Z -7.1667, A 0.000, B 0.000, C 0.000 }
gfCNCPoint5[24373] = {X 334.2270, Y 3.2503, Z -7.1667, A 0.000, B 0.000, C 0.000 }
gfCNCPoint5[24374] = {X 335.9775, Y 2.4248, Z -7.1667, A 0.000, B 0.000, C 0.000 }
gfCNCPoint5[24375] = {X 338.0600, Y 1.6135, Z -7.1667, A 0.000, B 0.000, C 0.000 }
gfCNCPoint5[24376] = {X 340.2043, Y 0.9836, Z -7.1667, A 0.000, B 0.000, C 0.000 }
gfCNCPoint5[24377] = {X 342.3947, Y 0.5395, Z -7.1667, A 0.000, B 0.000, C 0.000 }
gfCNCPoint5[24378] = {X 344.6151, Y 0.2846, Z -7.1667, A 0.000, B 0.000, C 0.000 }
gfCNCPoint5[24379] = {X 346.8491, Y 0.2208, Z -7.1667, A 0.000, B 0.000, C 0.000 }
gfCNCPoint5[24380] = {X 349.0804, Y 0.3485, Z -7.1667, A 0.000, B 0.000, C 0.000 }
gfCNCPoint5[24381] = {X 351.2926, Y 0.6668, Z -7.1667, A 0.000, B 0.000, C 0.000 }
gfCNCPoint5[24382] = {X 351.5598, Y 0.7170, Z -7.1667, A 0.000, B 0.000, C 0.000 }
gfCNCPoint5[24383] = {X 352.2984, Y -3.2142, Z -7.1667, A 0.000, B 0.000, C 0.000 }
gfCNCPoint5[24384] = {X 351.5450, Y 0.7956, Z -7.1667, A 0.000, B 0.000, C 0.000 }
gfCNCPoint5[24385] = {X 351.8101, Y 0.8454, Z -7.1667, A 0.000, B 0.000, C 0.000 }
gfCNCPoint5[24386] = {X 353.8990, Y 1.3806, Z -7.1667, A 0.000, B 0.000, C 0.000 }
gfCNCPoint5[24387] = {X 355.9210, Y 2.1301, Z -7.1667, A 0.000, B 0.000, C 0.000 }
gfCNCPoint5[24388] = {X 357.8541, Y 3.0858, Z -7.1667, A 0.000, B 0.000, C 0.000 }
gfCNCPoint5[24389] = {X 359.6772, Y 4.2374, Z -7.1667, A 0.000, B 0.000, C 0.000 }
gfCNCPoint5[24390] = {X 361.3707, Y 5.5724, Z -7.1667, A 0.000, B 0.000, C 0.000 }
gfCNCPoint5[24391] = {X 362.9162, Y 7.0763, Z -7.1667, A 0.000, B 0.000, C 0.000 }
gfCNCPoint5[24392] = {X 364.4421, Y 8.9219, Z -7.1667, A 0.000, B 0.000, C 0.000 }
gfCNCPoint5[24393] = {X 365.7809, Y 10.9076, Z -7.1667, A 0.000, B 0.000, C 0.000 }
gfCNCPoint5[24394] = {X 366.9196, Y 13.0142, Z -7.1667, A 0.000, B 0.000, C 0.000 }
gfCNCPoint5[24395] = {X 367.8476, Y 15.2219, Z -7.1667, A 0.000, B 0.000, C 0.000 }
gfCNCPoint5[24396] = {X 368.5559, Y 17.5095, Z -7.1667, A 0.000, B 0.000, C 0.000 }
gfCNCPoint5[24397] = {X 369.0329, Y 19.7787, Z -7.1667, A 0.000, B 0.000, C 0.000 }
gfCNCPoint5[24398] = {X 369.3405, Y 22.0769, Z -7.1667, A 0.000, B 0.000, C 0.000 }
gfCNCPoint5[24399] = {X 369.4769, Y 24.3917, Z -7.1667, A 0.000, B 0.000, C 0.000 }
gfCNCPoint5[24400] = {X 369.4414, Y 26.7102, Z -7.1667, A 0.000, B 0.000, C 0.000 }
gfCNCPoint5[24401] = {X 369.2342, Y 29.0196, Z -7.1667, A 0.000, B 0.000, C 0.000 }
gfCNCPoint5[24402] = {X 368.8564, Y 31.3074, Z -7.1667, A 0.000, B 0.000, C 0.000 }
gfCNCPoint5[24403] = {X 368.3391, Y 33.3846, Z -7.1667, A 0.000, B 0.000, C 0.000 }
gfCNCPoint5[24404] = {X 367.6403, Y 35.4079, Z -7.1667, A 0.000, B 0.000, C 0.000 }
gfCNCPoint5[24405] = {X 366.7656, Y 37.3617, Z -7.1667, A 0.000, B 0.000, C 0.000 }
gfCNCPoint5[24406] = {X 365.7217, Y 39.2305, Z -7.1667, A 0.000, B 0.000, C 0.000 }
gfCNCPoint5[24407] = {X 364.5169, Y 40.9999, Z -7.1667, A 0.000, B 0.000, C 0.000 }
gfCNCPoint5[24408] = {X 364.4010, Y 41.1583, Z -7.1667, A 0.000, B 0.000, C 0.000 }
gfCNCPoint5[24409] = {X 363.1253, Y 42.6975, Z -7.1667, A 0.000, B 0.000, C 0.000 }
gfCNCPoint5[24410] = {X 361.7132, Y 44.1124, Z -7.1667, A 0.000, B 0.000, C 0.000 }
gfCNCPoint5[24411] = {X 360.1767, Y 45.3913, Z -7.1667, A 0.000, B 0.000, C 0.000 }
gfCNCPoint5[24412] = {X 358.5288, Y 46.5230, Z -7.1667, A 0.000, B 0.000, C 0.000 }
gfCNCPoint5[24413] = {X 356.7837, Y 47.4980, Z -7.1667, A 0.000, B 0.000, C 0.000 }
gfCNCPoint5[24414] = {X 356.0912, Y 47.8259, Z -7.1667, A 0.000, B 0.000, C 0.000 }
gfCNCPoint5[24415] = {X 353.9238, Y 48.6345, Z -7.1667, A 0.000, B 0.000, C 0.000 }
gfCNCPoint5[24416] = {X 351.6854, Y 49.2183, Z -7.1667, A 0.000, B 0.000, C 0.000 }
gfCNCPoint5[24417] = {X 349.3992, Y 49.5714, Z -7.1667, A 0.000, B 0.000, C 0.000 }
gfCNCPoint5[24418] = {X 347.0889, Y 49.6899, Z -7.1667, A 0.000, B 0.000, C 0.000 }
gfCNCPoint5[24419] = {X 345.0499, Y 49.6559, Z -7.1667, A 0.000, B 0.000, C 0.000 }
gfCNCPoint5[24420] = {X 343.0216, Y 49.4451, Z -7.1667, A 0.000, B 0.000, C 0.000 }
gfCNCPoint5[24421] = {X 341.0191, Y 49.0592, Z -7.1667, A 0.000, B 0.000, C 0.000 }
gfCNCPoint5[24422] = {X 339.0577, Y 48.5011, Z -7.1667, A 0.000, B 0.000, C 0.000 }
gfCNCPoint5[24423] = {X 337.1521, Y 47.7749, Z -7.1667, A 0.000, B 0.000, C 0.000 }
gfCNCPoint5[24424] = {X 335.3167, Y 46.8862, Z -7.1667, A 0.000, B 0.000, C 0.000 }
gfCNCPoint5[24425] = {X 333.7137, Y 45.8936, Z -7.1667, A 0.000, B 0.000, C 0.000 }
gfCNCPoint5[24426] = {X 332.1953, Y 44.7761, Z -7.1667, A 0.000, B 0.000, C 0.000 }
gfCNCPoint5[24427] = {X 330.7711, Y 43.5406, Z -7.1667, A 0.000, B 0.000, C 0.000 }
gfCNCPoint5[24428] = {X 329.8559, Y 43.5681, Z -7.1667, A 0.000, B 0.000, C 0.000 }
gfCNCPoint5[24429] = {X 328.9584, Y 43.3867, Z -7.1667, A 0.000, B 0.000, C 0.000 }
gfCNCPoint5[24430] = {X 328.1256, Y 43.0060, Z -7.1667, A 0.000, B 0.000, C 0.000 }
gfCNCPoint5[24431] = {X 327.4013, Y 42.4458, Z -7.1667, A 0.000, B 0.000, C 0.000 }
gfCNCPoint5[24432] = {X 326.8042, Y 41.8634, Z -7.1667, A 0.000, B 0.000, C 0.000 }
gfCNCPoint5[24433] = {X 326.2223, Y 41.1472, Z -7.1667, A 0.000, B 0.000, C 0.000 }
gfCNCPoint5[24434] = {X 325.8201, Y 40.3166, Z -7.1667, A 0.000, B 0.000, C 0.000 }
gfCNCPoint5[24435] = {X 325.6189, Y 39.4160, Z -7.1667, A 0.000, B 0.000, C 0.000 }
gfCNCPoint5[24436] = {X 325.6294, Y 38.4932, Z -7.1667, A 0.000, B 0.000, C 0.000 }
gfCNCPoint5[24437] = {X 325.8511, Y 37.5974, Z -7.1667, A 0.000, B 0.000, C 0.000 }
gfCNCPoint5[24438] = {X 326.2722, Y 36.7763, Z -7.1667, A 0.000, B 0.000, C 0.000 }
gfCNCPoint5[24439] = {X 330.5290, Y 30.4119, Z -7.1667, A 0.000, B 0.000, C 0.000 }
gfCNCPoint5[24440] = {X 331.0932, Y 29.7536, Z -7.1667, A 0.000, B 0.000, C 0.000 }
gfCNCPoint5[24441] = {X 331.7861, Y 29.2322, Z -7.1667, A 0.000, B 0.000, C 0.000 }
gfCNCPoint5[24442] = {X 332.5750, Y 28.8725, Z -7.1667, A 0.000, B 0.000, C 0.000 }
gfCNCPoint5[24443] = {X 333.4229, Y 28.6911, Z -7.1667, A 0.000, B 0.000, C 0.000 }
gfCNCPoint5[24444] = {X 334.2900, Y 28.6968, Z -7.1667, A 0.000, B 0.000, C 0.000 }
gfCNCPoint5[24445] = {X 335.1355, Y 28.8892, Z -7.1667, A 0.000, B 0.000, C 0.000 }
gfCNCPoint5[24446] = {X 335.9196, Y 29.2593, Z -7.1667, A 0.000, B 0.000, C 0.000 }
gfCNCPoint5[24447] = {X 336.6056, Y 29.7896, Z -7.1667, A 0.000, B 0.000, C 0.000 }
gfCNCPoint5[24448] = {X 337.2041, Y 30.3665, Z -7.1667, A 0.000, B 0.000, C 0.000 }
gfCNCPoint5[24449] = {X 337.7863, Y 31.0895, Z -7.1667, A 0.000, B 0.000, C 0.000 }
gfCNCPoint5[24450] = {X 338.1862, Y 31.9272, Z -7.1667, A 0.000, B 0.000, C 0.000 }
gfCNCPoint5[24451] = {X 338.3822, Y 32.8346, Z -7.1667, A 0.000, B 0.000, C 0.000 }
gfCNCPoint5[24452] = {X 338.3638, Y 33.7627, Z -7.1667, A 0.000, B 0.000, C 0.000 }
gfCNCPoint5[24453] = {X 338.3475, Y 33.8705, Z -7.1667, A 0.000, B 0.000, C 0.000 }
gfCNCPoint5[24454] = {X 338.3283, Y 33.9779, Z -7.1667, A 0.000, B 0.000, C 0.000 }
gfCNCPoint5[24455] = {X 338.4902, Y 34.1122, Z -7.1667, A 0.000, B 0.000, C 0.000 }
gfCNCPoint5[24456] = {X 339.2774, Y 34.8319, Z -7.1667, A 0.000, B 0.000, C 0.000 }
gfCNCPoint5[24457] = {X 340.4116, Y 35.7390, Z -7.1667, A 0.000, B 0.000, C 0.000 }
gfCNCPoint5[24458] = {X 341.6553, Y 36.4889, Z -7.1667, A 0.000, B 0.000, C 0.000 }
gfCNCPoint5[24459] = {X 342.9869, Y 37.0684, Z -7.1667, A 0.000, B 0.000, C 0.000 }
gfCNCPoint5[24460] = {X 344.3833, Y 37.4676, Z -7.1667, A 0.000, B 0.000, C 0.000 }
gfCNCPoint5[24461] = {X 345.8201, Y 37.6795, Z -7.1667, A 0.000, B 0.000, C 0.000 }
gfCNCPoint5[24462] = {X 347.2722, Y 37.7003, Z -7.1667, A 0.000, B 0.000, C 0.000 }
gfCNCPoint5[24463] = {X 347.5354, Y 37.6867, Z -7.1667, A 0.000, B 0.000, C 0.000 }
gfCNCPoint5[24464] = {X 348.7320, Y 37.5459, Z -7.1667, A 0.000, B 0.000, C 0.000 }
gfCNCPoint5[24465] = {X 349.9000, Y 37.2501, Z -7.1667, A 0.000, B 0.000, C 0.000 }
gfCNCPoint5[24466] = {X 351.0194, Y 36.8045, Z -7.1667, A 0.000, B 0.000, C 0.000 }
gfCNCPoint5[24467] = {X 352.0711, Y 36.2166, Z -7.1667, A 0.000, B 0.000, C 0.000 }
gfCNCPoint5[24468] = {X 353.0371, Y 35.4966, Z -7.1667, A 0.000, B 0.000, C 0.000 }
gfCNCPoint5[24469] = {X 354.2202, Y 34.3468, Z -7.1667, A 0.000, B 0.000, C 0.000 }
gfCNCPoint5[24470] = {X 355.2441, Y 33.0532, Z -7.1667, A 0.000, B 0.000, C 0.000 }
gfCNCPoint5[24471] = {X 356.0914, Y 31.6377, Z -7.1667, A 0.000, B 0.000, C 0.000 }
gfCNCPoint5[24472] = {X 356.7477, Y 30.1241, Z -7.1667, A 0.000, B 0.000, C 0.000 }
gfCNCPoint5[24473] = {X 357.2020, Y 28.5381, Z -7.1667, A 0.000, B 0.000, C 0.000 }
gfCNCPoint5[24474] = {X 357.4803, Y 26.8196, Z -7.1667, A 0.000, B 0.000, C 0.000 }
gfCNCPoint5[24475] = {X 357.5936, Y 25.0823, Z -7.1667, A 0.000, B 0.000, C 0.000 }
gfCNCPoint5[24476] = {X 357.5411, Y 23.3422, Z -7.1667, A 0.000, B 0.000, C 0.000 }
gfCNCPoint5[24477] = {X 357.3231, Y 21.6150, Z -7.1667, A 0.000, B 0.000, C 0.000 }
gfCNCPoint5[24478] = {X 356.9597, Y 20.0590, Z -7.1667, A 0.000, B 0.000, C 0.000 }
gfCNCPoint5[24479] = {X 356.3954, Y 18.5642, Z -7.1667, A 0.000, B 0.000, C 0.000 }
gfCNCPoint5[24480] = {X 355.6399, Y 17.1563, Z -7.1667, A 0.000, B 0.000, C 0.000 }
gfCNCPoint5[24481] = {X 354.7062, Y 15.8596, Z -7.1667, A 0.000, B 0.000, C 0.000 }
gfCNCPoint5[24482] = {X 353.8052, Y 14.9007, Z -7.1667, A 0.000, B 0.000, C 0.000 }
gfCNCPoint5[24483] = {X 352.7800, Y 14.0758, Z -7.1667, A 0.000, B 0.000, C 0.000 }
gfCNCPoint5[24484] = {X 351.6502, Y 13.4011, Z -7.1667, A 0.000, B 0.000, C 0.000 }
gfCNCPoint5[24485] = {X 350.4379, Y 12.8895, Z -7.1667, A 0.000, B 0.000, C 0.000 }
gfCNCPoint5[24486] = {X 349.1664, Y 12.5509, Z -7.1667, A 0.000, B 0.000, C 0.000 }
gfCNCPoint5[24487] = {X 347.3712, Y 12.3261, Z -7.1667, A 0.000, B 0.000, C 0.000 }
gfCNCPoint5[24488] = {X 345.5620, Y 12.3402, Z -7.1667, A 0.000, B 0.000, C 0.000 }
gfCNCPoint5[24489] = {X 343.7706, Y 12.5928, Z -7.1667, A 0.000, B 0.000, C 0.000 }
gfCNCPoint5[24490] = {X 342.0281, Y 13.0797, Z -7.1667, A 0.000, B 0.000, C 0.000 }
gfCNCPoint5[24491] = {X 340.3651, Y 13.7922, Z -7.1667, A 0.000, B 0.000, C 0.000 }
gfCNCPoint5[24492] = {X 338.8107, Y 14.7179, Z -7.1667, A 0.000, B 0.000, C 0.000 }
gfCNCPoint5[24493] = {X 338.7182, Y 14.7822, Z -7.1667, A 0.000, B 0.000, C 0.000 }
gfCNCPoint5[24494] = {X 338.6262, Y 14.8472, Z -7.1667, A 0.000, B 0.000, C 0.000 }
gfCNCPoint5[24495] = {X 338.6380, Y 15.0639, Z -7.1667, A 0.000, B 0.000, C 0.000 }
gfCNCPoint5[24496] = {X 338.5595, Y 16.0361, Z -7.1667, A 0.000, B 0.000, C 0.000 }
gfCNCPoint5[24497] = {X 338.2481, Y 16.9605, Z -7.1667, A 0.000, B 0.000, C 0.000 }
gfCNCPoint5[24498] = {X 337.7223, Y 17.7819, Z -7.1667, A 0.000, B 0.000, C 0.000 }
gfCNCPoint5[24499] = {X 337.0132, Y 18.4517, Z -7.1667, A 0.000, B 0.000, C 0.000 }
gfCNCPoint5[24500] = {X 336.3278, Y 18.9560, Z -7.1667, A 0.000, B 0.000, C 0.000 }
gfCNCPoint5[24501] = {X 335.5713, Y 19.3817, Z -7.1667, A 0.000, B 0.000, C 0.000 }
gfCNCPoint5[24502] = {X 334.7407, Y 19.6341, Z -7.1667, A 0.000, B 0.000, C 0.000 }
gfCNCPoint5[24503] = {X 333.8753, Y 19.7014, Z -7.1667, A 0.000, B 0.000, C 0.000 }
gfCNCPoint5[24504] = {X 333.0157, Y 19.5804, Z -7.1667, A 0.000, B 0.000, C 0.000 }
gfCNCPoint5[24505] = {X 332.2025, Y 19.2768, Z -7.1667, A 0.000, B 0.000, C 0.000 }
gfCNCPoint5[24506] = {X 331.4739, Y 18.8049, Z -7.1667, A 0.000, B 0.000, C 0.000 }
gfCNCPoint5[24507] = {X 330.8643, Y 18.1870, Z -7.1667, A 0.000, B 0.000, C 0.000 }
gfCNCPoint5[24508] = {X 330.4023, Y 17.4521, Z -7.1667, A 0.000, B 0.000, C 0.000 }
gfCNCPoint5[24509] = {X 326.8820, Y 10.2103, Z -7.1667, A 0.000, B 0.000, C 0.000 }
gfCNCPoint5[24510] = {X 326.5719, Y 9.3163, Z -7.1667, A 0.000, B 0.000, C 0.000 }
gfCNCPoint5[24511] = {X 326.4804, Y 8.3746, Z -7.1667, A 0.000, B 0.000, C 0.000 }
gfCNCPoint5[24512] = {X 326.6127, Y 7.4376, Z -7.1667, A 0.000, B 0.000, C 0.000 }
gfCNCPoint5[24513] = {X 326.9614, Y 6.5580, Z -7.1667, A 0.000, B 0.000, C 0.000 }
gfCNCPoint5[24514] = {X 327.5070, Y 5.7849, Z -7.1667, A 0.000, B 0.000, C 0.000 }
gfCNCPoint5[24515] = {X 328.2189, Y 5.1616, Z -7.1667, A 0.000, B 0.000, C 0.000 }
gfCNCPoint5[24516] = {X 328.8880, Y 4.7034, Z -7.1667, A 0.000, B 0.000, C 0.000 }
gfCNCPoint5[24517] = {X 329.7043, Y 4.2813, Z -7.1667, A 0.000, B 0.000, C 0.000 }
gfCNCPoint5[24518] = {X 330.5954, Y 4.0567, Z -7.1667, A 0.000, B 0.000, C 0.000 }
gfCNCPoint5[24519] = {X 331.5142, Y 4.0413, Z -7.1667, A 0.000, B 0.000, C 0.000 }
gfCNCPoint5[24520] = {X 332.4122, Y 4.2361, Z -7.1667, A 0.000, B 0.000, C 0.000 }
gfCNCPoint5[24521] = {X 332.5467, Y 4.2811, Z -7.1667, A 0.000, B 0.000, C 0.000 }
gfCNCPoint5[24522] = {X 332.6252, Y 4.2338, Z -7.1667, A 0.000, B 0.000, C 0.000 }
gfCNCPoint5[24523] = {X 332.7038, Y 4.1867, Z -7.1667, A 0.000, B 0.000, C 0.000 }
gfCNCPoint5[24524] = {X 334.3287, Y 3.2881, Z -7.1667, A 0.000, B 0.000, C 0.000 }
gfCNCPoint5[24525] = {X 336.0092, Y 2.4982, Z -7.1667, A 0.000, B 0.000, C 0.000 }
gfCNCPoint5[24526] = {X 336.1736, Y 2.4272, Z -7.1667, A 0.000, B 0.000, C 0.000 }
gfCNCPoint5[24527] = {X 338.2310, Y 1.6408, Z -7.1667, A 0.000, B 0.000, C 0.000 }
gfCNCPoint5[24528] = {X 340.3476, Y 1.0313, Z -7.1667, A 0.000, B 0.000, C 0.000 }
gfCNCPoint5[24529] = {X 342.5081, Y 0.6031, Z -7.1667, A 0.000, B 0.000, C 0.000 }
gfCNCPoint5[24530] = {X 344.6972, Y 0.3594, Z -7.1667, A 0.000, B 0.000, C 0.000 }
gfCNCPoint5[24531] = {X 346.8990, Y 0.3018, Z -7.1667, A 0.000, B 0.000, C 0.000 }
gfCNCPoint5[24532] = {X 349.0978, Y 0.4308, Z -7.1667, A 0.000, B 0.000, C 0.000 }
gfCNCPoint5[24533] = {X 351.2778, Y 0.7454, Z -7.1667, A 0.000, B 0.000, C 0.000 }
gfCNCPoint5[24534] = {X 351.5450, Y 0.7956, Z -7.1667, A 0.000, B 0.000, C 0.000 }
gfCNCPoint5[24535] = {X 352.2984, Y -3.2142, Z -7.1667, A 0.000, B 0.000, C 0.000 }
gfCNCPoint5[24536] = {X 352.2984, Y -3.2142, Z -4.1667, A 0.000, B 0.000, C 0.000 }
gfCNCPoint5[24537] = {X 352.2984, Y -3.2142, Z 11.0000, A 0.000, B 0.000, C 0.000 }
gfCNCPoint5[24538] = {X 606.0426, Y 42.9004, Z 11.0000, A 0.000, B 0.000, C 0.000 }
gfCNCPoint5[24539] = {X 606.0426, Y 42.9004, Z -4.1667, A 0.000, B 0.000, C 0.000 }
gfCNCPoint5[24540] = {X 606.0426, Y 42.9004, Z -7.1667, A 0.000, B 0.000, C 0.000 }
gfCNCPoint5[24541] = {X 603.6967, Y 47.0766, Z -7.1667, A 0.000, B 0.000, C 0.000 }
gfCNCPoint5[24542] = {X 603.6312, Y 47.1891, Z -7.1667, A 0.000, B 0.000, C 0.000 }
gfCNCPoint5[24543] = {X 603.5622, Y 47.2996, Z -7.1667, A 0.000, B 0.000, C 0.000 }
gfCNCPoint5[24544] = {X 603.0358, Y 47.9600, Z -7.1667, A 0.000, B 0.000, C 0.000 }
gfCNCPoint5[24545] = {X 602.3890, Y 48.5029, Z -7.1667, A 0.000, B 0.000, C 0.000 }
gfCNCPoint5[24546] = {X 601.6473, Y 48.9069, Z -7.1667, A 0.000, B 0.000, C 0.000 }
gfCNCPoint5[24547] = {X 600.8403, Y 49.1559, Z -7.1667, A 0.000, B 0.000, C 0.000 }
gfCNCPoint5[24548] = {X 600.0000, Y 49.2400, Z -7.1667, A 0.000, B 0.000, C 0.000 }
gfCNCPoint5[24549] = {X 593.5565, Y 49.2400, Z -7.1667, A 0.000, B 0.000, C 0.000 }
gfCNCPoint5[24550] = {X 592.6130, Y 49.1337, Z -7.1667, A 0.000, B 0.000, C 0.000 }
gfCNCPoint5[24551] = {X 591.7169, Y 48.8201, Z -7.1667, A 0.000, B 0.000, C 0.000 }
gfCNCPoint5[24552] = {X 590.9129, Y 48.3150, Z -7.1667, A 0.000, B 0.000, C 0.000 }
gfCNCPoint5[24553] = {X 590.2416, Y 47.6436, Z -7.1667, A 0.000, B 0.000, C 0.000 }
gfCNCPoint5[24554] = {X 589.7364, Y 46.8397, Z -7.1667, A 0.000, B 0.000, C 0.000 }
gfCNCPoint5[24555] = {X 589.4228, Y 45.9435, Z -7.1667, A 0.000, B 0.000, C 0.000 }
gfCNCPoint5[24556] = {X 589.3165, Y 45.0000, Z -7.1667, A 0.000, B 0.000, C 0.000 }
gfCNCPoint5[24557] = {X 589.3165, Y 44.0650, Z -7.1667, A 0.000, B 0.000, C 0.000 }
gfCNCPoint5[24558] = {X 589.4204, Y 43.1448, Z -7.1667, A 0.000, B 0.000, C 0.000 }
gfCNCPoint5[24559] = {X 589.7199, Y 42.2685, Z -7.1667, A 0.000, B 0.000, C 0.000 }
gfCNCPoint5[24560] = {X 590.2010, Y 41.4771, Z -7.1667, A 0.000, B 0.000, C 0.000 }
gfCNCPoint5[24561] = {X 590.8412, Y 40.8079, Z -7.1667, A 0.000, B 0.000, C 0.000 }
gfCNCPoint5[24562] = {X 590.8420, Y 33.1224, Z -7.1667, A 0.000, B 0.000, C 0.000 }
gfCNCPoint5[24563] = {X 585.3714, Y 46.6218, Z -7.1667, A 0.000, B 0.000, C 0.000 }
gfCNCPoint5[24564] = {X 585.0085, Y 47.3114, Z -7.1667, A 0.000, B 0.000, C 0.000 }
gfCNCPoint5[24565] = {X 584.5255, Y 47.9228, Z -7.1667, A 0.000, B 0.000, C 0.000 }
gfCNCPoint5[24566] = {X 583.9387, Y 48.4356, Z -7.1667, A 0.000, B 0.000, C 0.000 }
gfCNCPoint5[24567] = {X 583.2680, Y 48.8323, Z -7.1667, A 0.000, B 0.000, C 0.000 }
gfCNCPoint5[24568] = {X 582.3418, Y 49.1460, Z -7.1667, A 0.000, B 0.000, C 0.000 }
gfCNCPoint5[24569] = {X 581.3682, Y 49.2391, Z -7.1667, A 0.000, B 0.000, C 0.000 }
gfCNCPoint5[24570] = {X 580.3993, Y 49.1068, Z -7.1667, A 0.000, B 0.000, C 0.000 }
gfCNCPoint5[24571] = {X 579.4864, Y 48.7559, Z -7.1667, A 0.000, B 0.000, C 0.000 }
gfCNCPoint5[24572] = {X 578.6782, Y 48.2052, Z -7.1667, A 0.000, B 0.000, C 0.000 }
gfCNCPoint5[24573] = {X 578.0177, Y 47.4840, Z -7.1667, A 0.000, B 0.000, C 0.000 }
gfCNCPoint5[24574] = {X 577.5400, Y 46.6307, Z -7.1667, A 0.000, B 0.000, C 0.000 }
gfCNCPoint5[24575] = {X 571.9399, Y 32.9370, Z -7.1667, A 0.000, B 0.000, C 0.000 }
gfCNCPoint5[24576] = {X 571.9401, Y 40.8086, Z -7.1667, A 0.000, B 0.000, C 0.000 }
gfCNCPoint5[24577] = {X 572.5776, Y 41.4689, Z -7.1667, A 0.000, B 0.000, C 0.000 }
gfCNCPoint5[24578] = {X 573.0580, Y 42.2509, Z -7.1667, A 0.000, B 0.000, C 0.000 }
gfCNCPoint5[24579] = {X 573.3590, Y 43.1179, Z -7.1667, A 0.000, B 0.000, C 0.000 }
gfCNCPoint5[24580] = {X 573.4663, Y 44.0294, Z -7.1667, A 0.000, B 0.000, C 0.000 }
gfCNCPoint5[24581] = {X 573.4664, Y 45.0000, Z -7.1667, A 0.000, B 0.000, C 0.000 }
gfCNCPoint5[24582] = {X 573.3601, Y 45.9435, Z -7.1667, A 0.000, B 0.000, C 0.000 }
gfCNCPoint5[24583] = {X 573.0465, Y 46.8397, Z -7.1667, A 0.000, B 0.000, C 0.000 }
gfCNCPoint5[24584] = {X 572.5414, Y 47.6436, Z -7.1667, A 0.000, B 0.000, C 0.000 }
gfCNCPoint5[24585] = {X 571.8700, Y 48.3150, Z -7.1667, A 0.000, B 0.000, C 0.000 }
gfCNCPoint5[24586] = {X 571.0661, Y 48.8201, Z -7.1667, A 0.000, B 0.000, C 0.000 }
gfCNCPoint5[24587] = {X 570.1699, Y 49.1337, Z -7.1667, A 0.000, B 0.000, C 0.000 }
gfCNCPoint5[24588] = {X 569.2264, Y 49.2400, Z -7.1667, A 0.000, B 0.000, C 0.000 }
gfCNCPoint5[24589] = {X 562.4443, Y 49.2400, Z -7.1667, A 0.000, B 0.000, C 0.000 }
gfCNCPoint5[24590] = {X 561.5008, Y 49.1337, Z -7.1667, A 0.000, B 0.000, C 0.000 }
gfCNCPoint5[24591] = {X 560.6046, Y 48.8201, Z -7.1667, A 0.000, B 0.000, C 0.000 }
gfCNCPoint5[24592] = {X 559.8007, Y 48.3150, Z -7.1667, A 0.000, B 0.000, C 0.000 }
gfCNCPoint5[24593] = {X 559.1293, Y 47.6436, Z -7.1667, A 0.000, B 0.000, C 0.000 }
gfCNCPoint5[24594] = {X 558.6242, Y 46.8397, Z -7.1667, A 0.000, B 0.000, C 0.000 }
gfCNCPoint5[24595] = {X 558.3106, Y 45.9435, Z -7.1667, A 0.000, B 0.000, C 0.000 }
gfCNCPoint5[24596] = {X 558.2043, Y 45.0000, Z -7.1667, A 0.000, B 0.000, C 0.000 }
gfCNCPoint5[24597] = {X 558.2043, Y 44.0652, Z -7.1667, A 0.000, B 0.000, C 0.000 }
gfCNCPoint5[24598] = {X 558.3079, Y 43.1444, Z -7.1667, A 0.000, B 0.000, C 0.000 }
gfCNCPoint5[24599] = {X 558.6078, Y 42.2677, Z -7.1667, A 0.000, B 0.000, C 0.000 }
gfCNCPoint5[24600] = {X 559.0896, Y 41.4763, Z -7.1667, A 0.000, B 0.000, C 0.000 }
gfCNCPoint5[24601] = {X 559.7309, Y 40.8076, Z -7.1667, A 0.000, B 0.000, C 0.000 }
gfCNCPoint5[24602] = {X 559.7310, Y 9.1922, Z -7.1667, A 0.000, B 0.000, C 0.000 }
gfCNCPoint5[24603] = {X 559.0934, Y 8.5319, Z -7.1667, A 0.000, B 0.000, C 0.000 }
gfCNCPoint5[24604] = {X 558.6128, Y 7.7499, Z -7.1667, A 0.000, B 0.000, C 0.000 }
gfCNCPoint5[24605] = {X 558.3118, Y 6.8827, Z -7.1667, A 0.000, B 0.000, C 0.000 }
gfCNCPoint5[24606] = {X 558.2045, Y 5.9711, Z -7.1667, A 0.000, B 0.000, C 0.000 }
gfCNCPoint5[24607] = {X 558.2043, Y 5.0000, Z -7.1667, A 0.000, B 0.000, C 0.000 }
gfCNCPoint5[24608] = {X 558.3106, Y 4.0565, Z -7.1667, A 0.000, B 0.000, C 0.000 }
gfCNCPoint5[24609] = {X 558.6242, Y 3.1603, Z -7.1667, A 0.000, B 0.000, C 0.000 }
gfCNCPoint5[24610] = {X 559.1293, Y 2.3564, Z -7.1667, A 0.000, B 0.000, C 0.000 }
gfCNCPoint5[24611] = {X 559.8007, Y 1.6850, Z -7.1667, A 0.000, B 0.000, C 0.000 }
gfCNCPoint5[24612] = {X 560.6046, Y 1.1799, Z -7.1667, A 0.000, B 0.000, C 0.000 }
gfCNCPoint5[24613] = {X 561.5008, Y 0.8663, Z -7.1667, A 0.000, B 0.000, C 0.000 }
gfCNCPoint5[24614] = {X 562.4443, Y 0.7600, Z -7.1667, A 0.000, B 0.000, C 0.000 }
gfCNCPoint5[24615] = {X 570.9376, Y 0.7600, Z -7.1667, A 0.000, B 0.000, C 0.000 }
gfCNCPoint5[24616] = {X 571.8810, Y 0.8663, Z -7.1667, A 0.000, B 0.000, C 0.000 }
gfCNCPoint5[24617] = {X 572.7772, Y 1.1799, Z -7.1667, A 0.000, B 0.000, C 0.000 }
gfCNCPoint5[24618] = {X 573.5812, Y 1.6850, Z -7.1667, A 0.000, B 0.000, C 0.000 }
gfCNCPoint5[24619] = {X 574.2525, Y 2.3564, Z -7.1667, A 0.000, B 0.000, C 0.000 }
gfCNCPoint5[24620] = {X 574.7577, Y 3.1603, Z -7.1667, A 0.000, B 0.000, C 0.000 }
gfCNCPoint5[24621] = {X 575.0712, Y 4.0565, Z -7.1667, A 0.000, B 0.000, C 0.000 }
gfCNCPoint5[24622] = {X 575.1776, Y 5.0000, Z -7.1667, A 0.000, B 0.000, C 0.000 }
gfCNCPoint5[24623] = {X 575.1776, Y 5.9343, Z -7.1667, A 0.000, B 0.000, C 0.000 }
gfCNCPoint5[24624] = {X 575.1024, Y 6.7287, Z -7.1667, A 0.000, B 0.000, C 0.000 }
gfCNCPoint5[24625] = {X 574.8797, Y 7.4951, Z -7.1667, A 0.000, B 0.000, C 0.000 }
gfCNCPoint5[24626] = {X 574.5174, Y 8.2061, Z -7.1667, A 0.000, B 0.000, C 0.000 }
gfCNCPoint5[24627] = {X 581.1908, Y 24.5805, Z -7.1667, A 0.000, B 0.000, C 0.000 }
gfCNCPoint5[24628] = {X 587.9345, Y 8.0875, Z -7.1667, A 0.000, B 0.000, C 0.000 }
gfCNCPoint5[24629] = {X 587.6157, Y 7.4196, Z -7.1667, A 0.000, B 0.000, C 0.000 }
gfCNCPoint5[24630] = {X 587.4179, Y 6.7065, Z -7.1667, A 0.000, B 0.000, C 0.000 }
gfCNCPoint5[24631] = {X 587.3471, Y 5.9698, Z -7.1667, A 0.000, B 0.000, C 0.000 }
gfCNCPoint5[24632] = {X 587.3470, Y 5.0000, Z -7.1667, A 0.000, B 0.000, C 0.000 }
gfCNCPoint5[24633] = {X 587.4533, Y 4.0565, Z -7.1667, A 0.000, B 0.000, C 0.000 }
gfCNCPoint5[24634] = {X 587.7668, Y 3.1603, Z -7.1667, A 0.000, B 0.000, C 0.000 }
gfCNCPoint5[24635] = {X 588.2720, Y 2.3564, Z -7.1667, A 0.000, B 0.000, C 0.000 }
gfCNCPoint5[24636] = {X 588.9434, Y 1.6850, Z -7.1667, A 0.000, B 0.000, C 0.000 }
gfCNCPoint5[24637] = {X 589.7473, Y 1.1799, Z -7.1667, A 0.000, B 0.000, C 0.000 }
gfCNCPoint5[24638] = {X 590.6435, Y 0.8663, Z -7.1667, A 0.000, B 0.000, C 0.000 }
gfCNCPoint5[24639] = {X 591.5870, Y 0.7600, Z -7.1667, A 0.000, B 0.000, C 0.000 }
gfCNCPoint5[24640] = {X 600.0000, Y 0.7600, Z -7.1667, A 0.000, B 0.000, C 0.000 }
gfCNCPoint5[24641] = {X 600.8403, Y 0.8441, Z -7.1667, A 0.000, B 0.000, C 0.000 }
gfCNCPoint5[24642] = {X 601.6473, Y 1.0931, Z -7.1667, A 0.000, B 0.000, C 0.000 }
gfCNCPoint5[24643] = {X 602.3890, Y 1.4971, Z -7.1667, A 0.000, B 0.000, C 0.000 }
gfCNCPoint5[24644] = {X 603.0358, Y 2.0400, Z -7.1667, A 0.000, B 0.000, C 0.000 }
gfCNCPoint5[24645] = {X 603.5622, Y 2.7004, Z -7.1667, A 0.000, B 0.000, C 0.000 }
gfCNCPoint5[24646] = {X 603.6312, Y 2.8109, Z -7.1667, A 0.000, B 0.000, C 0.000 }
gfCNCPoint5[24647] = {X 603.6967, Y 2.9234, Z -7.1667, A 0.000, B 0.000, C 0.000 }
gfCNCPoint5[24648] = {X 607.8226, Y 10.2681, Z -7.1667, A 0.000, B 0.000, C 0.000 }
gfCNCPoint5[24649] = {X 607.8226, Y 10.2681, Z -4.1667, A 0.000, B 0.000, C 0.000 }
gfCNCPoint5[24650] = {X 607.8226, Y 10.2681, Z 11.0000, A 0.000, B 0.000, C 0.000 }
gfCNCPoint5[24651] = {X 607.6967, Y 39.1579, Z 11.0000, A 0.000, B 0.000, C 0.000 }
gfCNCPoint5[24652] = {X 607.6967, Y 39.1579, Z -4.1667, A 0.000, B 0.000, C 0.000 }
gfCNCPoint5[24653] = {X 607.6967, Y 39.1579, Z -7.1667, A 0.000, B 0.000, C 0.000 }
gfCNCPoint5[24654] = {X 603.6967, Y 46.9079, Z -7.1667, A 0.000, B 0.000, C 0.000 }
gfCNCPoint5[24655] = {X 603.6001, Y 47.0845, Z -7.1667, A 0.000, B 0.000, C 0.000 }
gfCNCPoint5[24656] = {X 603.4950, Y 47.2562, Z -7.1667, A 0.000, B 0.000, C 0.000 }
gfCNCPoint5[24657] = {X 602.9785, Y 47.9041, Z -7.1667, A 0.000, B 0.000, C 0.000 }
gfCNCPoint5[24658] = {X 602.3439, Y 48.4368, Z -7.1667, A 0.000, B 0.000, C 0.000 }
gfCNCPoint5[24659] = {X 601.6162, Y 48.8332, Z -7.1667, A 0.000, B 0.000, C 0.000 }
gfCNCPoint5[24660] = {X 600.8245, Y 49.0775, Z -7.1667, A 0.000, B 0.000, C 0.000 }
gfCNCPoint5[24661] = {X 600.0000, Y 49.1600, Z -7.1667, A 0.000, B 0.000, C 0.000 }
gfCNCPoint5[24662] = {X 593.5565, Y 49.1600, Z -7.1667, A 0.000, B 0.000, C 0.000 }
gfCNCPoint5[24663] = {X 592.6308, Y 49.0557, Z -7.1667, A 0.000, B 0.000, C 0.000 }
gfCNCPoint5[24664] = {X 591.7516, Y 48.7480, Z -7.1667, A 0.000, B 0.000, C 0.000 }
gfCNCPoint5[24665] = {X 590.9628, Y 48.2524, Z -7.1667, A 0.000, B 0.000, C 0.000 }
gfCNCPoint5[24666] = {X 590.3041, Y 47.5937, Z -7.1667, A 0.000, B 0.000, C 0.000 }
gfCNCPoint5[24667] = {X 589.8085, Y 46.8050, Z -7.1667, A 0.000, B 0.000, C 0.000 }
gfCNCPoint5[24668] = {X 589.5008, Y 45.9257, Z -7.1667, A 0.000, B 0.000, C 0.000 }
gfCNCPoint5[24669] = {X 589.3965, Y 45.0000, Z -7.1667, A 0.000, B 0.000, C 0.000 }
gfCNCPoint5[24670] = {X 589.3965, Y 44.0653, Z -7.1667, A 0.000, B 0.000, C 0.000 }
gfCNCPoint5[24671] = {X 589.5005, Y 43.1533, Z -7.1667, A 0.000, B 0.000, C 0.000 }
gfCNCPoint5[24672] = {X 589.8003, Y 42.2856, Z -7.1667, A 0.000, B 0.000, C 0.000 }
gfCNCPoint5[24673] = {X 590.2815, Y 41.5038, Z -7.1667, A 0.000, B 0.000, C 0.000 }
gfCNCPoint5[24674] = {X 590.9212, Y 40.8454, Z -7.1667, A 0.000, B 0.000, C 0.000 }
gfCNCPoint5[24675] = {X 590.9220, Y 32.7119, Z -7.1667, A 0.000, B 0.000, C 0.000 }
gfCNCPoint5[24676] = {X 585.2975, Y 46.5912, Z -7.1667, A 0.000, B 0.000, C 0.000 }
gfCNCPoint5[24677] = {X 584.9414, Y 47.2678, Z -7.1667, A 0.000, B 0.000, C 0.000 }
gfCNCPoint5[24678] = {X 584.4675, Y 47.8677, Z -7.1667, A 0.000, B 0.000, C 0.000 }
gfCNCPoint5[24679] = {X 583.8918, Y 48.3708, Z -7.1667, A 0.000, B 0.000, C 0.000 }
gfCNCPoint5[24680] = {X 583.2338, Y 48.7600, Z -7.1667, A 0.000, B 0.000, C 0.000 }
gfCNCPoint5[24681] = {X 582.3250, Y 49.0678, Z -7.1667, A 0.000, B 0.000, C 0.000 }
gfCNCPoint5[24682] = {X 581.3699, Y 49.1592, Z -7.1667, A 0.000, B 0.000, C 0.000 }
gfCNCPoint5[24683] = {X 580.4192, Y 49.0293, Z -7.1667, A 0.000, B 0.000, C 0.000 }
gfCNCPoint5[24684] = {X 579.5236, Y 48.6850, Z -7.1667, A 0.000, B 0.000, C 0.000 }
gfCNCPoint5[24685] = {X 578.7306, Y 48.1448, Z -7.1667, A 0.000, B 0.000, C 0.000 }
gfCNCPoint5[24686] = {X 578.0826, Y 47.4372, Z -7.1667, A 0.000, B 0.000, C 0.000 }
gfCNCPoint5[24687] = {X 577.6138, Y 46.5999, Z -7.1667, A 0.000, B 0.000, C 0.000 }
gfCNCPoint5[24688] = {X 571.8599, Y 32.5300, Z -7.1667, A 0.000, B 0.000, C 0.000 }
gfCNCPoint5[24689] = {X 571.8601, Y 40.8463, Z -7.1667, A 0.000, B 0.000, C 0.000 }
gfCNCPoint5[24690] = {X 572.4971, Y 41.4958, Z -7.1667, A 0.000, B 0.000, C 0.000 }
gfCNCPoint5[24691] = {X 572.9777, Y 42.2683, Z -7.1667, A 0.000, B 0.000, C 0.000 }
gfCNCPoint5[24692] = {X 573.2789, Y 43.1267, Z -7.1667, A 0.000, B 0.000, C 0.000 }
gfCNCPoint5[24693] = {X 573.3863, Y 44.0301, Z -7.1667, A 0.000, B 0.000, C 0.000 }
gfCNCPoint5[24694] = {X 573.3864, Y 45.0000, Z -7.1667, A 0.000, B 0.000, C 0.000 }
gfCNCPoint5[24695] = {X 573.2821, Y 45.9257, Z -7.1667, A 0.000, B 0.000, C 0.000 }
gfCNCPoint5[24696] = {X 572.9745, Y 46.8050, Z -7.1667, A 0.000, B 0.000, C 0.000 }
gfCNCPoint5[24697] = {X 572.4788, Y 47.5937, Z -7.1667, A 0.000, B 0.000, C 0.000 }
gfCNCPoint5[24698] = {X 571.8201, Y 48.2524, Z -7.1667, A 0.000, B 0.000, C 0.000 }
gfCNCPoint5[24699] = {X 571.0314, Y 48.7480, Z -7.1667, A 0.000, B 0.000, C 0.000 }
gfCNCPoint5[24700] = {X 570.1521, Y 49.0557, Z -7.1667, A 0.000, B 0.000, C 0.000 }
gfCNCPoint5[24701] = {X 569.2264, Y 49.1600, Z -7.1667, A 0.000, B 0.000, C 0.000 }
gfCNCPoint5[24702] = {X 562.4443, Y 49.1600, Z -7.1667, A 0.000, B 0.000, C 0.000 }
gfCNCPoint5[24703] = {X 561.5186, Y 49.0557, Z -7.1667, A 0.000, B 0.000, C 0.000 }
gfCNCPoint5[24704] = {X 560.6393, Y 48.7480, Z -7.1667, A 0.000, B 0.000, C 0.000 }
gfCNCPoint5[24705] = {X 559.8506, Y 48.2524, Z -7.1667, A 0.000, B 0.000, C 0.000 }
gfCNCPoint5[24706] = {X 559.1919, Y 47.5937, Z -7.1667, A 0.000, B 0.000, C 0.000 }
gfCNCPoint5[24707] = {X 558.6963, Y 46.8050, Z -7.1667, A 0.000, B 0.000, C 0.000 }
gfCNCPoint5[24708] = {X 558.3886, Y 45.9257, Z -7.1667, A 0.000, B 0.000, C 0.000 }
gfCNCPoint5[24709] = {X 558.2843, Y 45.0000, Z -7.1667, A 0.000, B 0.000, C 0.000 }
gfCNCPoint5[24710] = {X 558.2843, Y 44.0654, Z -7.1667, A 0.000, B 0.000, C 0.000 }
gfCNCPoint5[24711] = {X 558.3880, Y 43.1529, Z -7.1667, A 0.000, B 0.000, C 0.000 }
gfCNCPoint5[24712] = {X 558.6881, Y 42.2849, Z -7.1667, A 0.000, B 0.000, C 0.000 }
gfCNCPoint5[24713] = {X 559.1701, Y 41.5031, Z -7.1667, A 0.000, B 0.000, C 0.000 }
gfCNCPoint5[24714] = {X 559.8109, Y 40.8451, Z -7.1667, A 0.000, B 0.000, C 0.000 }
gfCNCPoint5[24715] = {X 559.8110, Y 9.1545, Z -7.1667, A 0.000, B 0.000, C 0.000 }
gfCNCPoint5[24716] = {X 559.1739, Y 8.5050, Z -7.1667, A 0.000, B 0.000, C 0.000 }
gfCNCPoint5[24717] = {X 558.6931, Y 7.7325, Z -7.1667, A 0.000, B 0.000, C 0.000 }
gfCNCPoint5[24718] = {X 558.3919, Y 6.8739, Z -7.1667, A 0.000, B 0.000, C 0.000 }
gfCNCPoint5[24719] = {X 558.2845, Y 5.9704, Z -7.1667, A 0.000, B 0.000, C 0.000 }
gfCNCPoint5[24720] = {X 558.2843, Y 5.0000, Z -7.1667, A 0.000, B 0.000, C 0.000 }
gfCNCPoint5[24721] = {X 558.3886, Y 4.0743, Z -7.1667, A 0.000, B 0.000, C 0.000 }
gfCNCPoint5[24722] = {X 558.6963, Y 3.1950, Z -7.1667, A 0.000, B 0.000, C 0.000 }
gfCNCPoint5[24723] = {X 559.1919, Y 2.4063, Z -7.1667, A 0.000, B 0.000, C 0.000 }
gfCNCPoint5[24724] = {X 559.8506, Y 1.7476, Z -7.1667, A 0.000, B 0.000, C 0.000 }
gfCNCPoint5[24725] = {X 560.6393, Y 1.2520, Z -7.1667, A 0.000, B 0.000, C 0.000 }
gfCNCPoint5[24726] = {X 561.5186, Y 0.9443, Z -7.1667, A 0.000, B 0.000, C 0.000 }
gfCNCPoint5[24727] = {X 562.4443, Y 0.8400, Z -7.1667, A 0.000, B 0.000, C 0.000 }
gfCNCPoint5[24728] = {X 570.9376, Y 0.8400, Z -7.1667, A 0.000, B 0.000, C 0.000 }
gfCNCPoint5[24729] = {X 571.8632, Y 0.9443, Z -7.1667, A 0.000, B 0.000, C 0.000 }
gfCNCPoint5[24730] = {X 572.7425, Y 1.2520, Z -7.1667, A 0.000, B 0.000, C 0.000 }
gfCNCPoint5[24731] = {X 573.5313, Y 1.7476, Z -7.1667, A 0.000, B 0.000, C 0.000 }
gfCNCPoint5[24732] = {X 574.1900, Y 2.4063, Z -7.1667, A 0.000, B 0.000, C 0.000 }
gfCNCPoint5[24733] = {X 574.6856, Y 3.1950, Z -7.1667, A 0.000, B 0.000, C 0.000 }
gfCNCPoint5[24734] = {X 574.9933, Y 4.0743, Z -7.1667, A 0.000, B 0.000, C 0.000 }
gfCNCPoint5[24735] = {X 575.0976, Y 5.0000, Z -7.1667, A 0.000, B 0.000, C 0.000 }
gfCNCPoint5[24736] = {X 575.0976, Y 5.9343, Z -7.1667, A 0.000, B 0.000, C 0.000 }
gfCNCPoint5[24737] = {X 575.0212, Y 6.7272, Z -7.1667, A 0.000, B 0.000, C 0.000 }
gfCNCPoint5[24738] = {X 574.7952, Y 7.4911, Z -7.1667, A 0.000, B 0.000, C 0.000 }
gfCNCPoint5[24739] = {X 574.4277, Y 8.1979, Z -7.1667, A 0.000, B 0.000, C 0.000 }
gfCNCPoint5[24740] = {X 581.1907, Y 24.7921, Z -7.1667, A 0.000, B 0.000, C 0.000 }
gfCNCPoint5[24741] = {X 588.0237, Y 8.0808, Z -7.1667, A 0.000, B 0.000, C 0.000 }
gfCNCPoint5[24742] = {X 587.7000, Y 7.4162, Z -7.1667, A 0.000, B 0.000, C 0.000 }
gfCNCPoint5[24743] = {X 587.4990, Y 6.7049, Z -7.1667, A 0.000, B 0.000, C 0.000 }
gfCNCPoint5[24744] = {X 587.4271, Y 5.9692, Z -7.1667, A 0.000, B 0.000, C 0.000 }
gfCNCPoint5[24745] = {X 587.4270, Y 5.0000, Z -7.1667, A 0.000, B 0.000, C 0.000 }
gfCNCPoint5[24746] = {X 587.5313, Y 4.0743, Z -7.1667, A 0.000, B 0.000, C 0.000 }
gfCNCPoint5[24747] = {X 587.8389, Y 3.1950, Z -7.1667, A 0.000, B 0.000, C 0.000 }
gfCNCPoint5[24748] = {X 588.3345, Y 2.4063, Z -7.1667, A 0.000, B 0.000, C 0.000 }
gfCNCPoint5[24749] = {X 588.9932, Y 1.7476, Z -7.1667, A 0.000, B 0.000, C 0.000 }
gfCNCPoint5[24750] = {X 589.7820, Y 1.2520, Z -7.1667, A 0.000, B 0.000, C 0.000 }
gfCNCPoint5[24751] = {X 590.6613, Y 0.9443, Z -7.1667, A 0.000, B 0.000, C 0.000 }
gfCNCPoint5[24752] = {X 591.5870, Y 0.8400, Z -7.1667, A 0.000, B 0.000, C 0.000 }
gfCNCPoint5[24753] = {X 600.0000, Y 0.8400, Z -7.1667, A 0.000, B 0.000, C 0.000 }
gfCNCPoint5[24754] = {X 600.8245, Y 0.9225, Z -7.1667, A 0.000, B 0.000, C 0.000 }
gfCNCPoint5[24755] = {X 601.6162, Y 1.1668, Z -7.1667, A 0.000, B 0.000, C 0.000 }
gfCNCPoint5[24756] = {X 602.3439, Y 1.5632, Z -7.1667, A 0.000, B 0.000, C 0.000 }
gfCNCPoint5[24757] = {X 602.9785, Y 2.0959, Z -7.1667, A 0.000, B 0.000, C 0.000 }
gfCNCPoint5[24758] = {X 603.4950, Y 2.7438, Z -7.1667, A 0.000, B 0.000, C 0.000 }
gfCNCPoint5[24759] = {X 603.6001, Y 2.9155, Z -7.1667, A 0.000, B 0.000, C 0.000 }
gfCNCPoint5[24760] = {X 603.6967, Y 3.0921, Z -7.1667, A 0.000, B 0.000, C 0.000 }
gfCNCPoint5[24761] = {X 607.6967, Y 10.8421, Z -7.1667, A 0.000, B 0.000, C 0.000 }
gfCNCPoint5[24762] = {X 607.6967, Y 10.8421, Z -4.1667, A 0.000, B 0.000, C 0.000 }
gfCNCPoint5[24763] = {X 607.6967, Y 10.8421, Z 11.0000, A 0.000, B 0.000, C 0.000 }
gfCNCPoint5[24764] = {X 607.6967, Y 38.1624, Z 11.0000, A 0.000, B 0.000, C 0.000 }
gfCNCPoint5[24765] = {X 607.6967, Y 38.1624, Z -4.1667, A 0.000, B 0.000, C 0.000 }
gfCNCPoint5[24766] = {X 607.6967, Y 38.1624, Z -7.1667, A 0.000, B 0.000, C 0.000 }
gfCNCPoint5[24767] = {X 603.6967, Y 46.7266, Z -7.1667, A 0.000, B 0.000, C 0.000 }
gfCNCPoint5[24768] = {X 603.5705, Y 46.9743, Z -7.1667, A 0.000, B 0.000, C 0.000 }
gfCNCPoint5[24769] = {X 603.4278, Y 47.2128, Z -7.1667, A 0.000, B 0.000, C 0.000 }
gfCNCPoint5[24770] = {X 602.9213, Y 47.8483, Z -7.1667, A 0.000, B 0.000, C 0.000 }
gfCNCPoint5[24771] = {X 602.2988, Y 48.3707, Z -7.1667, A 0.000, B 0.000, C 0.000 }
gfCNCPoint5[24772] = {X 601.5852, Y 48.7595, Z -7.1667, A 0.000, B 0.000, C 0.000 }
gfCNCPoint5[24773] = {X 600.8086, Y 48.9991, Z -7.1667, A 0.000, B 0.000, C 0.000 }
gfCNCPoint5[24774] = {X 600.0000, Y 49.0800, Z -7.1667, A 0.000, B 0.000, C 0.000 }
gfCNCPoint5[24775] = {X 593.5565, Y 49.0800, Z -7.1667, A 0.000, B 0.000, C 0.000 }
gfCNCPoint5[24776] = {X 592.6486, Y 48.9777, Z -7.1667, A 0.000, B 0.000, C 0.000 }
gfCNCPoint5[24777] = {X 591.7863, Y 48.6760, Z -7.1667, A 0.000, B 0.000, C 0.000 }
gfCNCPoint5[24778] = {X 591.0127, Y 48.1899, Z -7.1667, A 0.000, B 0.000, C 0.000 }
gfCNCPoint5[24779] = {X 590.3667, Y 47.5438, Z -7.1667, A 0.000, B 0.000, C 0.000 }
gfCNCPoint5[24780] = {X 589.8806, Y 46.7702, Z -7.1667, A 0.000, B 0.000, C 0.000 }
gfCNCPoint5[24781] = {X 589.5788, Y 45.9079, Z -7.1667, A 0.000, B 0.000, C 0.000 }
gfCNCPoint5[24782] = {X 589.4765, Y 45.0000, Z -7.1667, A 0.000, B 0.000, C 0.000 }
gfCNCPoint5[24783] = {X 589.4765, Y 44.0657, Z -7.1667, A 0.000, B 0.000, C 0.000 }
gfCNCPoint5[24784] = {X 589.5806, Y 43.1618, Z -7.1667, A 0.000, B 0.000, C 0.000 }
gfCNCPoint5[24785] = {X 589.8807, Y 42.3029, Z -7.1667, A 0.000, B 0.000, C 0.000 }
gfCNCPoint5[24786] = {X 590.3620, Y 41.5308, Z -7.1667, A 0.000, B 0.000, C 0.000 }
gfCNCPoint5[24787] = {X 591.0012, Y 40.8833, Z -7.1667, A 0.000, B 0.000, C 0.000 }
gfCNCPoint5[24788] = {X 591.0021, Y 32.3014, Z -7.1667, A 0.000, B 0.000, C 0.000 }
gfCNCPoint5[24789] = {X 585.2236, Y 46.5606, Z -7.1667, A 0.000, B 0.000, C 0.000 }
gfCNCPoint5[24790] = {X 584.8743, Y 47.2242, Z -7.1667, A 0.000, B 0.000, C 0.000 }
gfCNCPoint5[24791] = {X 584.4095, Y 47.8125, Z -7.1667, A 0.000, B 0.000, C 0.000 }
gfCNCPoint5[24792] = {X 583.8449, Y 48.3059, Z -7.1667, A 0.000, B 0.000, C 0.000 }
gfCNCPoint5[24793] = {X 583.1996, Y 48.6877, Z -7.1667, A 0.000, B 0.000, C 0.000 }
gfCNCPoint5[24794] = {X 582.3082, Y 48.9895, Z -7.1667, A 0.000, B 0.000, C 0.000 }
gfCNCPoint5[24795] = {X 581.3715, Y 49.0792, Z -7.1667, A 0.000, B 0.000, C 0.000 }
gfCNCPoint5[24796] = {X 580.4391, Y 48.9518, Z -7.1667, A 0.000, B 0.000, C 0.000 }
gfCNCPoint5[24797] = {X 579.5607, Y 48.6142, Z -7.1667, A 0.000, B 0.000, C 0.000 }
gfCNCPoint5[24798] = {X 578.7830, Y 48.0843, Z -7.1667, A 0.000, B 0.000, C 0.000 }
gfCNCPoint5[24799] = {X 578.1474, Y 47.3903, Z -7.1667, A 0.000, B 0.000, C 0.000 }
gfCNCPoint5[24800] = {X 577.6877, Y 46.5692, Z -7.1667, A 0.000, B 0.000, C 0.000 }
gfCNCPoint5[24801] = {X 571.7799, Y 32.1230, Z -7.1667, A 0.000, B 0.000, C 0.000 }
gfCNCPoint5[24802] = {X 571.7801, Y 40.8840, Z -7.1667, A 0.000, B 0.000, C 0.000 }
gfCNCPoint5[24803] = {X 571.8686, Y 40.9571, Z -7.1667, A 0.000, B 0.000, C 0.000 }
gfCNCPoint5[24804] = {X 572.4697, Y 41.5905, Z -7.1667, A 0.000, B 0.000, C 0.000 }
gfCNCPoint5[24805] = {X 572.9222, Y 42.3374, Z -7.1667, A 0.000, B 0.000, C 0.000 }
gfCNCPoint5[24806] = {X 573.2054, Y 43.1634, Z -7.1667, A 0.000, B 0.000, C 0.000 }
gfCNCPoint5[24807] = {X 573.3063, Y 44.0308, Z -7.1667, A 0.000, B 0.000, C 0.000 }
gfCNCPoint5[24808] = {X 573.3064, Y 45.0000, Z -7.1667, A 0.000, B 0.000, C 0.000 }
gfCNCPoint5[24809] = {X 573.2041, Y 45.9079, Z -7.1667, A 0.000, B 0.000, C 0.000 }
gfCNCPoint5[24810] = {X 572.9024, Y 46.7702, Z -7.1667, A 0.000, B 0.000, C 0.000 }
gfCNCPoint5[24811] = {X 572.4163, Y 47.5438, Z -7.1667, A 0.000, B 0.000, C 0.000 }
gfCNCPoint5[24812] = {X 571.7703, Y 48.1899, Z -7.1667, A 0.000, B 0.000, C 0.000 }
gfCNCPoint5[24813] = {X 570.9967, Y 48.6760, Z -7.1667, A 0.000, B 0.000, C 0.000 }
gfCNCPoint5[24814] = {X 570.1343, Y 48.9777, Z -7.1667, A 0.000, B 0.000, C 0.000 }
gfCNCPoint5[24815] = {X 569.2264, Y 49.0800, Z -7.1667, A 0.000, B 0.000, C 0.000 }
gfCNCPoint5[24816] = {X 562.4443, Y 49.0800, Z -7.1667, A 0.000, B 0.000, C 0.000 }
gfCNCPoint5[24817] = {X 561.5364, Y 48.9777, Z -7.1667, A 0.000, B 0.000, C 0.000 }
gfCNCPoint5[24818] = {X 560.6741, Y 48.6760, Z -7.1667, A 0.000, B 0.000, C 0.000 }
gfCNCPoint5[24819] = {X 559.9005, Y 48.1899, Z -7.1667, A 0.000, B 0.000, C 0.000 }
gfCNCPoint5[24820] = {X 559.2544, Y 47.5438, Z -7.1667, A 0.000, B 0.000, C 0.000 }
gfCNCPoint5[24821] = {X 558.7683, Y 46.7702, Z -7.1667, A 0.000, B 0.000, C 0.000 }
gfCNCPoint5[24822] = {X 558.4666, Y 45.9079, Z -7.1667, A 0.000, B 0.000, C 0.000 }
gfCNCPoint5[24823] = {X 558.3643, Y 45.0000, Z -7.1667, A 0.000, B 0.000, C 0.000 }
gfCNCPoint5[24824] = {X 558.3643, Y 44.0657, Z -7.1667, A 0.000, B 0.000, C 0.000 }
gfCNCPoint5[24825] = {X 558.4603, Y 43.1965, Z -7.1667, A 0.000, B 0.000, C 0.000 }
gfCNCPoint5[24826] = {X 558.7380, Y 42.3673, Z -7.1667, A 0.000, B 0.000, C 0.000 }
gfCNCPoint5[24827] = {X 559.1848, Y 41.6156, Z -7.1667, A 0.000, B 0.000, C 0.000 }
gfCNCPoint5[24828] = {X 559.7806, Y 40.9754, Z -7.1667, A 0.000, B 0.000, C 0.000 }
gfCNCPoint5[24829] = {X 559.8353, Y 40.9288, Z -7.1667, A 0.000, B 0.000, C 0.000 }
gfCNCPoint5[24830] = {X 559.8909, Y 40.8831, Z -7.1667, A 0.000, B 0.000, C 0.000 }
gfCNCPoint5[24831] = {X 559.8910, Y 9.1164, Z -7.1667, A 0.000, B 0.000, C 0.000 }
gfCNCPoint5[24832] = {X 559.2543, Y 8.4778, Z -7.1667, A 0.000, B 0.000, C 0.000 }
gfCNCPoint5[24833] = {X 558.7735, Y 7.7149, Z -7.1667, A 0.000, B 0.000, C 0.000 }
gfCNCPoint5[24834] = {X 558.4719, Y 6.8651, Z -7.1667, A 0.000, B 0.000, C 0.000 }
gfCNCPoint5[24835] = {X 558.3645, Y 5.9697, Z -7.1667, A 0.000, B 0.000, C 0.000 }
gfCNCPoint5[24836] = {X 558.3643, Y 5.0000, Z -7.1667, A 0.000, B 0.000, C 0.000 }
gfCNCPoint5[24837] = {X 558.4666, Y 4.0921, Z -7.1667, A 0.000, B 0.000, C 0.000 }
gfCNCPoint5[24838] = {X 558.7683, Y 3.2298, Z -7.1667, A 0.000, B 0.000, C 0.000 }
gfCNCPoint5[24839] = {X 559.2544, Y 2.4562, Z -7.1667, A 0.000, B 0.000, C 0.000 }
gfCNCPoint5[24840] = {X 559.9005, Y 1.8101, Z -7.1667, A 0.000, B 0.000, C 0.000 }
gfCNCPoint5[24841] = {X 560.6741, Y 1.3240, Z -7.1667, A 0.000, B 0.000, C 0.000 }
gfCNCPoint5[24842] = {X 561.5364, Y 1.0223, Z -7.1667, A 0.000, B 0.000, C 0.000 }
gfCNCPoint5[24843] = {X 562.4443, Y 0.9200, Z -7.1667, A 0.000, B 0.000, C 0.000 }
gfCNCPoint5[24844] = {X 570.9376, Y 0.9200, Z -7.1667, A 0.000, B 0.000, C 0.000 }
gfCNCPoint5[24845] = {X 571.8454, Y 1.0223, Z -7.1667, A 0.000, B 0.000, C 0.000 }
gfCNCPoint5[24846] = {X 572.7078, Y 1.3240, Z -7.1667, A 0.000, B 0.000, C 0.000 }
gfCNCPoint5[24847] = {X 573.4814, Y 1.8101, Z -7.1667, A 0.000, B 0.000, C 0.000 }
gfCNCPoint5[24848] = {X 574.1274, Y 2.4562, Z -7.1667, A 0.000, B 0.000, C 0.000 }
gfCNCPoint5[24849] = {X 574.6135, Y 3.2298, Z -7.1667, A 0.000, B 0.000, C 0.000 }
gfCNCPoint5[24850] = {X 574.9153, Y 4.0921, Z -7.1667, A 0.000, B 0.000, C 0.000 }
gfCNCPoint5[24851] = {X 575.0176, Y 5.0000, Z -7.1667, A 0.000, B 0.000, C 0.000 }
gfCNCPoint5[24852] = {X 575.0176, Y 5.9342, Z -7.1667, A 0.000, B 0.000, C 0.000 }
gfCNCPoint5[24853] = {X 574.9500, Y 6.6732, Z -7.1667, A 0.000, B 0.000, C 0.000 }
gfCNCPoint5[24854] = {X 574.7498, Y 7.3877, Z -7.1667, A 0.000, B 0.000, C 0.000 }
gfCNCPoint5[24855] = {X 574.4235, Y 8.0542, Z -7.1667, A 0.000, B 0.000, C 0.000 }
gfCNCPoint5[24856] = {X 574.3790, Y 8.1256, Z -7.1667, A 0.000, B 0.000, C 0.000 }
gfCNCPoint5[24857] = {X 574.3331, Y 8.1961, Z -7.1667, A 0.000, B 0.000, C 0.000 }
gfCNCPoint5[24858] = {X 574.3597, Y 8.2419, Z -7.1667, A 0.000, B 0.000, C 0.000 }
gfCNCPoint5[24859] = {X 581.1906, Y 25.0038, Z -7.1667, A 0.000, B 0.000, C 0.000 }
gfCNCPoint5[24860] = {X 588.1130, Y 8.0737, Z -7.1667, A 0.000, B 0.000, C 0.000 }
gfCNCPoint5[24861] = {X 587.7843, Y 7.4126, Z -7.1667, A 0.000, B 0.000, C 0.000 }
gfCNCPoint5[24862] = {X 587.5801, Y 6.7031, Z -7.1667, A 0.000, B 0.000, C 0.000 }
gfCNCPoint5[24863] = {X 587.5071, Y 5.9685, Z -7.1667, A 0.000, B 0.000, C 0.000 }
gfCNCPoint5[24864] = {X 587.5070, Y 5.0000, Z -7.1667, A 0.000, B 0.000, C 0.000 }
gfCNCPoint5[24865] = {X 587.6092, Y 4.0921, Z -7.1667, A 0.000, B 0.000, C 0.000 }
gfCNCPoint5[24866] = {X 587.9110, Y 3.2298, Z -7.1667, A 0.000, B 0.000, C 0.000 }
gfCNCPoint5[24867] = {X 588.3971, Y 2.4562, Z -7.1667, A 0.000, B 0.000, C 0.000 }
gfCNCPoint5[24868] = {X 589.0431, Y 1.8101, Z -7.1667, A 0.000, B 0.000, C 0.000 }
gfCNCPoint5[24869] = {X 589.8167, Y 1.3240, Z -7.1667, A 0.000, B 0.000, C 0.000 }
gfCNCPoint5[24870] = {X 590.6791, Y 1.0223, Z -7.1667, A 0.000, B 0.000, C 0.000 }
gfCNCPoint5[24871] = {X 591.5870, Y 0.9200, Z -7.1667, A 0.000, B 0.000, C 0.000 }
gfCNCPoint5[24872] = {X 600.0000, Y 0.9200, Z -7.1667, A 0.000, B 0.000, C 0.000 }
gfCNCPoint5[24873] = {X 600.8086, Y 1.0009, Z -7.1667, A 0.000, B 0.000, C 0.000 }
gfCNCPoint5[24874] = {X 601.5852, Y 1.2405, Z -7.1667, A 0.000, B 0.000, C 0.000 }
gfCNCPoint5[24875] = {X 602.2988, Y 1.6293, Z -7.1667, A 0.000, B 0.000, C 0.000 }
gfCNCPoint5[24876] = {X 602.9213, Y 2.1517, Z -7.1667, A 0.000, B 0.000, C 0.000 }
gfCNCPoint5[24877] = {X 603.4278, Y 2.7872, Z -7.1667, A 0.000, B 0.000, C 0.000 }
gfCNCPoint5[24878] = {X 603.5705, Y 3.0257, Z -7.1667, A 0.000, B 0.000, C 0.000 }
gfCNCPoint5[24879] = {X 603.6967, Y 3.2734, Z -7.1667, A 0.000, B 0.000, C 0.000 }
gfCNCPoint5[24880] = {X 607.6967, Y 11.8376, Z -7.1667, A 0.000, B 0.000, C 0.000 }
gfCNCPoint5[24881] = {X 607.6967, Y 11.8376, Z -4.1667, A 0.000, B 0.000, C 0.000 }
gfCNCPoint5[24882] = {X 607.6967, Y 11.8376, Z 11.0000, A 0.000, B 0.000, C 0.000 }
gfCNCPoint5[24883] = {X 607.6967, Y 36.8506, Z 11.0000, A 0.000, B 0.000, C 0.000 }
gfCNCPoint5[24884] = {X 607.6967, Y 36.8506, Z -4.1667, A 0.000, B 0.000, C 0.000 }
gfCNCPoint5[24885] = {X 607.6967, Y 36.8506, Z -7.1667, A 0.000, B 0.000, C 0.000 }
gfCNCPoint5[24886] = {X 603.6967, Y 46.5280, Z -7.1667, A 0.000, B 0.000, C 0.000 }
gfCNCPoint5[24887] = {X 603.5432, Y 46.8563, Z -7.1667, A 0.000, B 0.000, C 0.000 }
gfCNCPoint5[24888] = {X 603.3606, Y 47.1694, Z -7.1667, A 0.000, B 0.000, C 0.000 }
gfCNCPoint5[24889] = {X 602.8640, Y 47.7924, Z -7.1667, A 0.000, B 0.000, C 0.000 }
gfCNCPoint5[24890] = {X 602.2537, Y 48.3046, Z -7.1667, A 0.000, B 0.000, C 0.000 }
gfCNCPoint5[24891] = {X 601.5541, Y 48.6858, Z -7.1667, A 0.000, B 0.000, C 0.000 }
gfCNCPoint5[24892] = {X 600.7928, Y 48.9207, Z -7.1667, A 0.000, B 0.000, C 0.000 }
gfCNCPoint5[24893] = {X 600.0000, Y 49.0000, Z -7.1667, A 0.000, B 0.000, C 0.000 }
gfCNCPoint5[24894] = {X 593.5565, Y 49.0000, Z -7.1667, A 0.000, B 0.000, C 0.000 }
gfCNCPoint5[24895] = {X 592.6664, Y 48.8997, Z -7.1667, A 0.000, B 0.000, C 0.000 }
gfCNCPoint5[24896] = {X 591.8210, Y 48.6039, Z -7.1667, A 0.000, B 0.000, C 0.000 }
gfCNCPoint5[24897] = {X 591.0626, Y 48.1273, Z -7.1667, A 0.000, B 0.000, C 0.000 }
gfCNCPoint5[24898] = {X 590.4292, Y 47.4940, Z -7.1667, A 0.000, B 0.000, C 0.000 }
gfCNCPoint5[24899] = {X 589.9527, Y 46.7355, Z -7.1667, A 0.000, B 0.000, C 0.000 }
gfCNCPoint5[24900] = {X 589.6568, Y 45.8901, Z -7.1667, A 0.000, B 0.000, C 0.000 }
gfCNCPoint5[24901] = {X 589.5565, Y 45.0000, Z -7.1667, A 0.000, B 0.000, C 0.000 }
gfCNCPoint5[24902] = {X 589.5565, Y 44.0660, Z -7.1667, A 0.000, B 0.000, C 0.000 }
gfCNCPoint5[24903] = {X 589.6607, Y 43.1704, Z -7.1667, A 0.000, B 0.000, C 0.000 }
gfCNCPoint5[24904] = {X 589.9611, Y 42.3203, Z -7.1667, A 0.000, B 0.000, C 0.000 }
gfCNCPoint5[24905] = {X 590.4425, Y 41.5581, Z -7.1667, A 0.000, B 0.000, C 0.000 }
gfCNCPoint5[24906] = {X 591.0811, Y 40.9217, Z -7.1667, A 0.000, B 0.000, C 0.000 }
gfCNCPoint5[24907] = {X 591.0821, Y 32.0441, Z -7.1667, A 0.000, B 0.000, C 0.000 }
gfCNCPoint5[24908] = {X 590.9675, Y 32.1736, Z -7.1667, A 0.000, B 0.000, C 0.000 }
gfCNCPoint5[24909] = {X 590.3112, Y 33.7933, Z -7.1667, A 0.000, B 0.000, C 0.000 }
gfCNCPoint5[24910] = {X 585.1497, Y 46.5300, Z -7.1667, A 0.000, B 0.000, C 0.000 }
gfCNCPoint5[24911] = {X 584.8073, Y 47.1805, Z -7.1667, A 0.000, B 0.000, C 0.000 }
gfCNCPoint5[24912] = {X 584.3516, Y 47.7574, Z -7.1667, A 0.000, B 0.000, C 0.000 }
gfCNCPoint5[24913] = {X 583.7980, Y 48.2411, Z -7.1667, A 0.000, B 0.000, C 0.000 }
gfCNCPoint5[24914] = {X 583.1653, Y 48.6154, Z -7.1667, A 0.000, B 0.000, C 0.000 }
gfCNCPoint5[24915] = {X 582.2878, Y 48.9121, Z -7.1667, A 0.000, B 0.000, C 0.000 }
gfCNCPoint5[24916] = {X 581.3656, Y 48.9990, Z -7.1667, A 0.000, B 0.000, C 0.000 }
gfCNCPoint5[24917] = {X 580.4481, Y 48.8715, Z -7.1667, A 0.000, B 0.000, C 0.000 }
gfCNCPoint5[24918] = {X 579.5845, Y 48.5363, Z -7.1667, A 0.000, B 0.000, C 0.000 }
gfCNCPoint5[24919] = {X 578.8212, Y 48.0115, Z -7.1667, A 0.000, B 0.000, C 0.000 }
gfCNCPoint5[24920] = {X 578.1990, Y 47.3251, Z -7.1667, A 0.000, B 0.000, C 0.000 }
gfCNCPoint5[24921] = {X 577.7515, Y 46.5141, Z -7.1667, A 0.000, B 0.000, C 0.000 }
gfCNCPoint5[24922] = {X 571.6998, Y 31.7160, Z -7.1667, A 0.000, B 0.000, C 0.000 }
gfCNCPoint5[24923] = {X 571.7001, Y 40.9217, Z -7.1667, A 0.000, B 0.000, C 0.000 }
gfCNCPoint5[24924] = {X 571.8389, Y 41.0369, Z -7.1667, A 0.000, B 0.000, C 0.000 }
gfCNCPoint5[24925] = {X 572.4244, Y 41.6633, Z -7.1667, A 0.000, B 0.000, C 0.000 }
gfCNCPoint5[24926] = {X 572.8630, Y 42.4001, Z -7.1667, A 0.000, B 0.000, C 0.000 }
gfCNCPoint5[24927] = {X 573.1345, Y 43.2134, Z -7.1667, A 0.000, B 0.000, C 0.000 }
gfCNCPoint5[24928] = {X 573.2264, Y 44.0660, Z -7.1667, A 0.000, B 0.000, C 0.000 }
gfCNCPoint5[24929] = {X 573.2264, Y 45.0000, Z -7.1667, A 0.000, B 0.000, C 0.000 }
gfCNCPoint5[24930] = {X 573.1261, Y 45.8901, Z -7.1667, A 0.000, B 0.000, C 0.000 }
gfCNCPoint5[24931] = {X 572.8303, Y 46.7355, Z -7.1667, A 0.000, B 0.000, C 0.000 }
gfCNCPoint5[24932] = {X 572.3538, Y 47.4940, Z -7.1667, A 0.000, B 0.000, C 0.000 }
gfCNCPoint5[24933] = {X 571.7204, Y 48.1273, Z -7.1667, A 0.000, B 0.000, C 0.000 }
gfCNCPoint5[24934] = {X 570.9620, Y 48.6039, Z -7.1667, A 0.000, B 0.000, C 0.000 }
gfCNCPoint5[24935] = {X 570.1165, Y 48.8997, Z -7.1667, A 0.000, B 0.000, C 0.000 }
gfCNCPoint5[24936] = {X 569.2264, Y 49.0000, Z -7.1667, A 0.000, B 0.000, C 0.000 }
gfCNCPoint5[24937] = {X 562.4443, Y 49.0000, Z -7.1667, A 0.000, B 0.000, C 0.000 }
gfCNCPoint5[24938] = {X 561.5542, Y 48.8997, Z -7.1667, A 0.000, B 0.000, C 0.000 }
gfCNCPoint5[24939] = {X 560.7088, Y 48.6039, Z -7.1667, A 0.000, B 0.000, C 0.000 }
gfCNCPoint5[24940] = {X 559.9503, Y 48.1273, Z -7.1667, A 0.000, B 0.000, C 0.000 }
gfCNCPoint5[24941] = {X 559.3170, Y 47.4940, Z -7.1667, A 0.000, B 0.000, C 0.000 }
gfCNCPoint5[24942] = {X 558.8404, Y 46.7355, Z -7.1667, A 0.000, B 0.000, C 0.000 }
gfCNCPoint5[24943] = {X 558.5446, Y 45.8901, Z -7.1667, A 0.000, B 0.000, C 0.000 }
gfCNCPoint5[24944] = {X 558.4443, Y 45.0000, Z -7.1667, A 0.000, B 0.000, C 0.000 }
gfCNCPoint5[24945] = {X 558.4443, Y 44.0660, Z -7.1667, A 0.000, B 0.000, C 0.000 }
gfCNCPoint5[24946] = {X 558.5384, Y 43.2137, Z -7.1667, A 0.000, B 0.000, C 0.000 }
gfCNCPoint5[24947] = {X 558.8107, Y 42.4006, Z -7.1667, A 0.000, B 0.000, C 0.000 }
gfCNCPoint5[24948] = {X 559.2488, Y 41.6635, Z -7.1667, A 0.000, B 0.000, C 0.000 }
gfCNCPoint5[24949] = {X 559.8330, Y 41.0359, Z -7.1667, A 0.000, B 0.000, C 0.000 }
gfCNCPoint5[24950] = {X 559.9013, Y 40.9779, Z -7.1667, A 0.000, B 0.000, C 0.000 }
gfCNCPoint5[24951] = {X 559.9709, Y 40.9215, Z -7.1667, A 0.000, B 0.000, C 0.000 }
gfCNCPoint5[24952] = {X 559.9710, Y 9.0778, Z -7.1667, A 0.000, B 0.000, C 0.000 }
gfCNCPoint5[24953] = {X 559.3293, Y 8.4434, Z -7.1667, A 0.000, B 0.000, C 0.000 }
gfCNCPoint5[24954] = {X 558.8462, Y 7.6814, Z -7.1667, A 0.000, B 0.000, C 0.000 }
gfCNCPoint5[24955] = {X 558.5460, Y 6.8305, Z -7.1667, A 0.000, B 0.000, C 0.000 }
gfCNCPoint5[24956] = {X 558.4443, Y 5.9340, Z -7.1667, A 0.000, B 0.000, C 0.000 }
gfCNCPoint5[24957] = {X 558.4443, Y 5.0000, Z -7.1667, A 0.000, B 0.000, C 0.000 }
gfCNCPoint5[24958] = {X 558.5446, Y 4.1099, Z -7.1667, A 0.000, B 0.000, C 0.000 }
gfCNCPoint5[24959] = {X 558.8404, Y 3.2645, Z -7.1667, A 0.000, B 0.000, C 0.000 }
gfCNCPoint5[24960] = {X 559.3170, Y 2.5060, Z -7.1667, A 0.000, B 0.000, C 0.000 }
gfCNCPoint5[24961] = {X 559.9503, Y 1.8727, Z -7.1667, A 0.000, B 0.000, C 0.000 }
gfCNCPoint5[24962] = {X 560.7088, Y 1.3961, Z -7.1667, A 0.000, B 0.000, C 0.000 }
gfCNCPoint5[24963] = {X 561.5542, Y 1.1003, Z -7.1667, A 0.000, B 0.000, C 0.000 }
gfCNCPoint5[24964] = {X 562.4443, Y 1.0000, Z -7.1667, A 0.000, B 0.000, C 0.000 }
gfCNCPoint5[24965] = {X 570.9376, Y 1.0000, Z -7.1667, A 0.000, B 0.000, C 0.000 }
gfCNCPoint5[24966] = {X 571.8276, Y 1.1003, Z -7.1667, A 0.000, B 0.000, C 0.000 }
gfCNCPoint5[24967] = {X 572.6731, Y 1.3961, Z -7.1667, A 0.000, B 0.000, C 0.000 }
gfCNCPoint5[24968] = {X 573.4315, Y 1.8727, Z -7.1667, A 0.000, B 0.000, C 0.000 }
gfCNCPoint5[24969] = {X 574.0649, Y 2.5060, Z -7.1667, A 0.000, B 0.000, C 0.000 }
gfCNCPoint5[24970] = {X 574.5414, Y 3.2645, Z -7.1667, A 0.000, B 0.000, C 0.000 }
gfCNCPoint5[24971] = {X 574.8373, Y 4.1099, Z -7.1667, A 0.000, B 0.000, C 0.000 }
gfCNCPoint5[24972] = {X 574.9376, Y 5.0000, Z -7.1667, A 0.000, B 0.000, C 0.000 }
gfCNCPoint5[24973] = {X 574.9372, Y 5.9858, Z -7.1667, A 0.000, B 0.000, C 0.000 }
gfCNCPoint5[24974] = {X 574.8650, Y 6.6925, Z -7.1667, A 0.000, B 0.000, C 0.000 }
gfCNCPoint5[24975] = {X 574.6689, Y 7.3753, Z -7.1667, A 0.000, B 0.000, C 0.000 }
gfCNCPoint5[24976] = {X 574.3551, Y 8.0126, Z -7.1667, A 0.000, B 0.000, C 0.000 }
gfCNCPoint5[24977] = {X 574.2922, Y 8.1127, Z -7.1667, A 0.000, B 0.000, C 0.000 }
gfCNCPoint5[24978] = {X 574.2264, Y 8.2108, Z -7.1667, A 0.000, B 0.000, C 0.000 }
gfCNCPoint5[24979] = {X 574.2619, Y 8.2359, Z -7.1667, A 0.000, B 0.000, C 0.000 }
gfCNCPoint5[24980] = {X 574.2857, Y 8.2723, Z -7.1667, A 0.000, B 0.000, C 0.000 }
gfCNCPoint5[24981] = {X 574.9161, Y 9.8068, Z -7.1667, A 0.000, B 0.000, C 0.000 }
gfCNCPoint5[24982] = {X 581.1904, Y 25.2156, Z -7.1667, A 0.000, B 0.000, C 0.000 }
gfCNCPoint5[24983] = {X 588.2025, Y 8.0661, Z -7.1667, A 0.000, B 0.000, C 0.000 }
gfCNCPoint5[24984] = {X 587.8646, Y 7.3983, Z -7.1667, A 0.000, B 0.000, C 0.000 }
gfCNCPoint5[24985] = {X 587.6570, Y 6.6792, Z -7.1667, A 0.000, B 0.000, C 0.000 }
gfCNCPoint5[24986] = {X 587.5870, Y 5.9340, Z -7.1667, A 0.000, B 0.000, C 0.000 }
gfCNCPoint5[24987] = {X 587.5870, Y 5.0000, Z -7.1667, A 0.000, B 0.000, C 0.000 }
gfCNCPoint5[24988] = {X 587.6872, Y 4.1099, Z -7.1667, A 0.000, B 0.000, C 0.000 }
gfCNCPoint5[24989] = {X 587.9831, Y 3.2645, Z -7.1667, A 0.000, B 0.000, C 0.000 }
gfCNCPoint5[24990] = {X 588.4596, Y 2.5060, Z -7.1667, A 0.000, B 0.000, C 0.000 }
gfCNCPoint5[24991] = {X 589.0930, Y 1.8727, Z -7.1667, A 0.000, B 0.000, C 0.000 }
gfCNCPoint5[24992] = {X 589.8514, Y 1.3961, Z -7.1667, A 0.000, B 0.000, C 0.000 }
gfCNCPoint5[24993] = {X 590.6969, Y 1.1003, Z -7.1667, A 0.000, B 0.000, C 0.000 }
gfCNCPoint5[24994] = {X 591.5870, Y 1.0000, Z -7.1667, A 0.000, B 0.000, C 0.000 }
gfCNCPoint5[24995] = {X 600.0000, Y 1.0000, Z -7.1667, A 0.000, B 0.000, C 0.000 }
gfCNCPoint5[24996] = {X 600.7928, Y 1.0793, Z -7.1667, A 0.000, B 0.000, C 0.000 }
gfCNCPoint5[24997] = {X 601.5541, Y 1.3142, Z -7.1667, A 0.000, B 0.000, C 0.000 }
gfCNCPoint5[24998] = {X 602.2537, Y 1.6954, Z -7.1667, A 0.000, B 0.000, C 0.000 }
gfCNCPoint5[24999] = {X 602.8640, Y 2.2076, Z -7.1667, A 0.000, B 0.000, C 0.000 }
gfCNCPoint5[25000] = {X 603.3606, Y 2.8306, Z -7.1667, A 0.000, B 0.000, C 0.000 }
gfCNCPoint5[25001] = {X 603.5432, Y 3.1437, Z -7.1667, A 0.000, B 0.000, C 0.000 }
gfCNCPoint5[25002] = {X 603.6967, Y 3.4720, Z -7.1667, A 0.000, B 0.000, C 0.000 }
gfCNCPoint5[25003] = {X 607.6967, Y 13.1494, Z -7.1667, A 0.000, B 0.000, C 0.000 }
gfCNCPoint5[25004] = {X 607.6967, Y 13.1494, Z -4.1667, A 0.000, B 0.000, C 0.000 }
gfCNCPoint5[25005] = {X 607.6967, Y 13.1494, Z 11.0000, A 0.000, B 0.000, C 0.000 }
gfCNCPoint5[25006] = {X 448.7153, Y 19.7827, Z 11.0000, A 0.000, B 0.000, C 0.000 }
gfCNCPoint5[25007] = {X 448.7153, Y 19.7827, Z -3.3333, A 0.000, B 0.000, C 0.000 }
gfCNCPoint5[25008] = {X 444.0414, Y 19.7828, Z -4.5857, A 0.000, B 0.000, C 0.000 }
gfCNCPoint5[25009] = {X 443.3486, Y 19.7990, Z -4.7714, A 0.000, B 0.000, C 0.000 }
gfCNCPoint5[25010] = {X 442.7492, Y 19.8056, Z -4.9320, A 0.000, B 0.000, C 0.000 }
gfCNCPoint5[25011] = {X 442.0369, Y 19.9289, Z -5.1257, A 0.000, B 0.000, C 0.000 }
gfCNCPoint5[25012] = {X 441.4701, Y 20.1240, Z -5.2863, A 0.000, B 0.000, C 0.000 }
gfCNCPoint5[25013] = {X 441.3672, Y 20.1595, Z -5.3155, A 0.000, B 0.000, C 0.000 }
gfCNCPoint5[25014] = {X 441.3343, Y 20.2632, Z -5.3446, A 0.000, B 0.000, C 0.000 }
gfCNCPoint5[25015] = {X 441.1896, Y 20.7191, Z -5.4728, A 0.000, B 0.000, C 0.000 }
gfCNCPoint5[25016] = {X 441.1560, Y 21.8873, Z -5.7860, A 0.000, B 0.000, C 0.000 }
gfCNCPoint5[25017] = {X 441.2742, Y 22.3508, Z -5.9141, A 0.000, B 0.000, C 0.000 }
gfCNCPoint5[25018] = {X 441.5045, Y 22.4261, Z -5.9790, A 0.000, B 0.000, C 0.000 }
gfCNCPoint5[25019] = {X 441.7458, Y 22.4478, Z -6.0440, A 0.000, B 0.000, C 0.000 }
gfCNCPoint5[25020] = {X 443.0153, Y 22.5622, Z -6.3855, A 0.000, B 0.000, C 0.000 }
gfCNCPoint5[25021] = {X 443.1164, Y 22.5663, Z -6.4126, A 0.000, B 0.000, C 0.000 }
gfCNCPoint5[25022] = {X 444.3942, Y 22.5560, Z -6.7550, A 0.000, B 0.000, C 0.000 }
gfCNCPoint5[25023] = {X 445.9305, Y 22.5560, Z -7.1667, A 0.000, B 0.000, C 0.000 }
gfCNCPoint5[25024] = {X 450.1184, Y 22.5560, Z -7.1667, A 0.000, B 0.000, C 0.000 }
gfCNCPoint5[25025] = {X 450.1184, Y 19.7826, Z -7.1667, A 0.000, B 0.000, C 0.000 }
gfCNCPoint5[25026] = {X 444.0414, Y 19.7828, Z -7.1667, A 0.000, B 0.000, C 0.000 }
gfCNCPoint5[25027] = {X 443.3486, Y 19.7990, Z -7.1667, A 0.000, B 0.000, C 0.000 }
gfCNCPoint5[25028] = {X 442.3963, Y 19.8861, Z -7.1667, A 0.000, B 0.000, C 0.000 }
gfCNCPoint5[25029] = {X 441.4701, Y 20.1240, Z -7.1667, A 0.000, B 0.000, C 0.000 }
gfCNCPoint5[25030] = {X 441.3857, Y 20.1775, Z -7.1667, A 0.000, B 0.000, C 0.000 }
gfCNCPoint5[25031] = {X 441.3343, Y 20.2632, Z -7.1667, A 0.000, B 0.000, C 0.000 }
gfCNCPoint5[25032] = {X 441.1844, Y 20.9513, Z -7.1667, A 0.000, B 0.000, C 0.000 }
gfCNCPoint5[25033] = {X 441.1642, Y 21.6552, Z -7.1667, A 0.000, B 0.000, C 0.000 }
gfCNCPoint5[25034] = {X 441.2742, Y 22.3508, Z -7.1667, A 0.000, B 0.000, C 0.000 }
gfCNCPoint5[25035] = {X 441.5072, Y 22.4127, Z -7.1667, A 0.000, B 0.000, C 0.000 }
gfCNCPoint5[25036] = {X 441.7458, Y 22.4478, Z -7.1667, A 0.000, B 0.000, C 0.000 }
gfCNCPoint5[25037] = {X 443.0687, Y 22.5344, Z -7.1667, A 0.000, B 0.000, C 0.000 }
gfCNCPoint5[25038] = {X 444.3942, Y 22.5560, Z -7.1667, A 0.000, B 0.000, C 0.000 }
gfCNCPoint5[25039] = {X 445.9305, Y 22.5560, Z -7.1667, A 0.000, B 0.000, C 0.000 }
gfCNCPoint5[25040] = {X 441.9457, Y 22.2874, Z -7.1667, A 0.000, B 0.000, C 0.000 }
gfCNCPoint5[25041] = {X 445.9305, Y 22.6360, Z -7.1667, A 0.000, B 0.000, C 0.000 }
gfCNCPoint5[25042] = {X 450.1984, Y 22.6360, Z -7.1667, A 0.000, B 0.000, C 0.000 }
gfCNCPoint5[25043] = {X 450.1984, Y 19.7026, Z -7.1667, A 0.000, B 0.000, C 0.000 }
gfCNCPoint5[25044] = {X 444.0404, Y 19.7028, Z -7.1667, A 0.000, B 0.000, C 0.000 }
gfCNCPoint5[25045] = {X 443.3497, Y 19.7189, Z -7.1667, A 0.000, B 0.000, C 0.000 }
gfCNCPoint5[25046] = {X 442.3836, Y 19.8071, Z -7.1667, A 0.000, B 0.000, C 0.000 }
gfCNCPoint5[25047] = {X 441.4441, Y 20.0484, Z -7.1667, A 0.000, B 0.000, C 0.000 }
gfCNCPoint5[25048] = {X 441.3285, Y 20.1216, Z -7.1667, A 0.000, B 0.000, C 0.000 }
gfCNCPoint5[25049] = {X 441.2581, Y 20.2390, Z -7.1667, A 0.000, B 0.000, C 0.000 }
gfCNCPoint5[25050] = {X 441.1033, Y 20.9560, Z -7.1667, A 0.000, B 0.000, C 0.000 }
gfCNCPoint5[25051] = {X 441.0863, Y 21.6893, Z -7.1667, A 0.000, B 0.000, C 0.000 }
gfCNCPoint5[25052] = {X 441.2077, Y 22.4128, Z -7.1667, A 0.000, B 0.000, C 0.000 }
gfCNCPoint5[25053] = {X 441.4696, Y 22.4865, Z -7.1667, A 0.000, B 0.000, C 0.000 }
gfCNCPoint5[25054] = {X 441.7387, Y 22.5275, Z -7.1667, A 0.000, B 0.000, C 0.000 }
gfCNCPoint5[25055] = {X 443.0645, Y 22.6143, Z -7.1667, A 0.000, B 0.000, C 0.000 }
gfCNCPoint5[25056] = {X 444.3930, Y 22.6360, Z -7.1667, A 0.000, B 0.000, C 0.000 }
gfCNCPoint5[25057] = {X 445.9305, Y 22.6360, Z -7.1667, A 0.000, B 0.000, C 0.000 }
gfCNCPoint5[25058] = {X 449.9153, Y 22.2874, Z -7.1667, A 0.000, B 0.000, C 0.000 }
gfCNCPoint5[25059] = {X 441.9457, Y 22.3674, Z -7.1667, A 0.000, B 0.000, C 0.000 }
gfCNCPoint5[25060] = {X 445.9305, Y 22.7160, Z -7.1667, A 0.000, B 0.000, C 0.000 }
gfCNCPoint5[25061] = {X 450.2784, Y 22.7160, Z -7.1667, A 0.000, B 0.000, C 0.000 }
gfCNCPoint5[25062] = {X 450.2784, Y 19.6226, Z -7.1667, A 0.000, B 0.000, C 0.000 }
gfCNCPoint5[25063] = {X 444.0395, Y 19.6228, Z -7.1667, A 0.000, B 0.000, C 0.000 }
gfCNCPoint5[25064] = {X 443.3483, Y 19.6390, Z -7.1667, A 0.000, B 0.000, C 0.000 }
gfCNCPoint5[25065] = {X 442.3698, Y 19.7283, Z -7.1667, A 0.000, B 0.000, C 0.000 }
gfCNCPoint5[25066] = {X 441.4180, Y 19.9727, Z -7.1667, A 0.000, B 0.000, C 0.000 }
gfCNCPoint5[25067] = {X 441.2712, Y 20.0657, Z -7.1667, A 0.000, B 0.000, C 0.000 }
gfCNCPoint5[25068] = {X 441.1818, Y 20.2148, Z -7.1667, A 0.000, B 0.000, C 0.000 }
gfCNCPoint5[25069] = {X 441.0222, Y 20.9605, Z -7.1667, A 0.000, B 0.000, C 0.000 }
gfCNCPoint5[25070] = {X 441.0086, Y 21.7230, Z -7.1667, A 0.000, B 0.000, C 0.000 }
gfCNCPoint5[25071] = {X 441.1414, Y 22.4740, Z -7.1667, A 0.000, B 0.000, C 0.000 }
gfCNCPoint5[25072] = {X 441.4321, Y 22.5601, Z -7.1667, A 0.000, B 0.000, C 0.000 }
gfCNCPoint5[25073] = {X 441.7315, Y 22.6072, Z -7.1667, A 0.000, B 0.000, C 0.000 }
gfCNCPoint5[25074] = {X 443.0611, Y 22.6942, Z -7.1667, A 0.000, B 0.000, C 0.000 }
gfCNCPoint5[25075] = {X 444.3933, Y 22.7160, Z -7.1667, A 0.000, B 0.000, C 0.000 }
gfCNCPoint5[25076] = {X 445.9305, Y 22.7160, Z -7.1667, A 0.000, B 0.000, C 0.000 }
gfCNCPoint5[25077] = {X 449.9153, Y 22.3674, Z -7.1667, A 0.000, B 0.000, C 0.000 }
gfCNCPoint5[25078] = {X 441.9457, Y 22.4474, Z -7.1667, A 0.000, B 0.000, C 0.000 }
gfCNCPoint5[25079] = {X 445.9305, Y 22.7960, Z -7.1667, A 0.000, B 0.000, C 0.000 }
gfCNCPoint5[25080] = {X 450.3584, Y 22.7960, Z -7.1667, A 0.000, B 0.000, C 0.000 }
gfCNCPoint5[25081] = {X 450.3584, Y 19.5426, Z -7.1667, A 0.000, B 0.000, C 0.000 }
gfCNCPoint5[25082] = {X 444.0385, Y 19.5428, Z -7.1667, A 0.000, B 0.000, C 0.000 }
gfCNCPoint5[25083] = {X 443.3469, Y 19.5590, Z -7.1667, A 0.000, B 0.000, C 0.000 }
gfCNCPoint5[25084] = {X 442.3559, Y 19.6495, Z -7.1667, A 0.000, B 0.000, C 0.000 }
gfCNCPoint5[25085] = {X 441.3920, Y 19.8971, Z -7.1667, A 0.000, B 0.000, C 0.000 }
gfCNCPoint5[25086] = {X 441.2140, Y 20.0099, Z -7.1667, A 0.000, B 0.000, C 0.000 }
gfCNCPoint5[25087] = {X 441.1056, Y 20.1906, Z -7.1667, A 0.000, B 0.000, C 0.000 }
gfCNCPoint5[25088] = {X 440.9412, Y 20.9648, Z -7.1667, A 0.000, B 0.000, C 0.000 }
gfCNCPoint5[25089] = {X 440.9311, Y 21.7563, Z -7.1667, A 0.000, B 0.000, C 0.000 }
gfCNCPoint5[25090] = {X 441.0755, Y 22.5345, Z -7.1667, A 0.000, B 0.000, C 0.000 }
gfCNCPoint5[25091] = {X 441.3945, Y 22.6336, Z -7.1667, A 0.000, B 0.000, C 0.000 }
gfCNCPoint5[25092] = {X 441.7243, Y 22.6869, Z -7.1667, A 0.000, B 0.000, C 0.000 }
gfCNCPoint5[25093] = {X 443.0576, Y 22.7741, Z -7.1667, A 0.000, B 0.000, C 0.000 }
gfCNCPoint5[25094] = {X 444.3936, Y 22.7960, Z -7.1667, A 0.000, B 0.000, C 0.000 }
gfCNCPoint5[25095] = {X 445.9305, Y 22.7960, Z -7.1667, A 0.000, B 0.000, C 0.000 }
gfCNCPoint5[25096] = {X 449.9153, Y 22.4474, Z -7.1667, A 0.000, B 0.000, C 0.000 }
gfCNCPoint5[25097] = {X 441.9457, Y 22.5274, Z -7.1667, A 0.000, B 0.000, C 0.000 }
gfCNCPoint5[25098] = {X 445.9305, Y 22.8760, Z -7.1667, A 0.000, B 0.000, C 0.000 }
gfCNCPoint5[25099] = {X 450.4384, Y 22.8760, Z -7.1667, A 0.000, B 0.000, C 0.000 }
gfCNCPoint5[25100] = {X 450.4384, Y 19.4626, Z -7.1667, A 0.000, B 0.000, C 0.000 }
gfCNCPoint5[25101] = {X 444.0376, Y 19.4628, Z -7.1667, A 0.000, B 0.000, C 0.000 }
gfCNCPoint5[25102] = {X 443.3456, Y 19.4790, Z -7.1667, A 0.000, B 0.000, C 0.000 }
gfCNCPoint5[25103] = {X 442.3420, Y 19.5707, Z -7.1667, A 0.000, B 0.000, C 0.000 }
gfCNCPoint5[25104] = {X 441.3660, Y 19.8215, Z -7.1667, A 0.000, B 0.000, C 0.000 }
gfCNCPoint5[25105] = {X 441.1567, Y 19.9540, Z -7.1667, A 0.000, B 0.000, C 0.000 }
gfCNCPoint5[25106] = {X 441.0293, Y 20.1664, Z -7.1667, A 0.000, B 0.000, C 0.000 }
gfCNCPoint5[25107] = {X 440.8603, Y 20.9690, Z -7.1667, A 0.000, B 0.000, C 0.000 }
gfCNCPoint5[25108] = {X 440.8537, Y 21.7892, Z -7.1667, A 0.000, B 0.000, C 0.000 }
gfCNCPoint5[25109] = {X 441.0097, Y 22.5944, Z -7.1667, A 0.000, B 0.000, C 0.000 }
gfCNCPoint5[25110] = {X 441.3570, Y 22.7068, Z -7.1667, A 0.000, B 0.000, C 0.000 }
gfCNCPoint5[25111] = {X 441.7172, Y 22.7665, Z -7.1667, A 0.000, B 0.000, C 0.000 }
gfCNCPoint5[25112] = {X 443.0542, Y 22.8540, Z -7.1667, A 0.000, B 0.000, C 0.000 }
gfCNCPoint5[25113] = {X 444.3939, Y 22.8760, Z -7.1667, A 0.000, B 0.000, C 0.000 }
gfCNCPoint5[25114] = {X 445.9305, Y 22.8760, Z -7.1667, A 0.000, B 0.000, C 0.000 }
gfCNCPoint5[25115] = {X 449.9153, Y 22.5274, Z -7.1667, A 0.000, B 0.000, C 0.000 }
gfCNCPoint5[25116] = {X 445.9305, Y 20.9560, Z -7.1667, A 0.000, B 0.000, C 0.000 }
gfCNCPoint5[25117] = {X 445.9305, Y 22.9560, Z -7.1667, A 0.000, B 0.000, C 0.000 }
gfCNCPoint5[25118] = {X 450.5184, Y 22.9560, Z -7.1667, A 0.000, B 0.000, C 0.000 }
gfCNCPoint5[25119] = {X 450.5184, Y 19.3826, Z -7.1667, A 0.000, B 0.000, C 0.000 }
gfCNCPoint5[25120] = {X 444.0367, Y 19.3828, Z -7.1667, A 0.000, B 0.000, C 0.000 }
gfCNCPoint5[25121] = {X 443.3442, Y 19.3990, Z -7.1667, A 0.000, B 0.000, C 0.000 }
gfCNCPoint5[25122] = {X 442.3281, Y 19.4919, Z -7.1667, A 0.000, B 0.000, C 0.000 }
gfCNCPoint5[25123] = {X 441.3399, Y 19.7458, Z -7.1667, A 0.000, B 0.000, C 0.000 }
gfCNCPoint5[25124] = {X 441.0995, Y 19.8981, Z -7.1667, A 0.000, B 0.000, C 0.000 }
gfCNCPoint5[25125] = {X 440.9531, Y 20.1422, Z -7.1667, A 0.000, B 0.000, C 0.000 }
gfCNCPoint5[25126] = {X 440.7794, Y 20.9730, Z -7.1667, A 0.000, B 0.000, C 0.000 }
gfCNCPoint5[25127] = {X 440.7764, Y 21.8217, Z -7.1667, A 0.000, B 0.000, C 0.000 }
gfCNCPoint5[25128] = {X 440.9441, Y 22.6537, Z -7.1667, A 0.000, B 0.000, C 0.000 }
gfCNCPoint5[25129] = {X 441.3195, Y 22.7800, Z -7.1667, A 0.000, B 0.000, C 0.000 }
gfCNCPoint5[25130] = {X 441.7100, Y 22.8462, Z -7.1667, A 0.000, B 0.000, C 0.000 }
gfCNCPoint5[25131] = {X 443.0508, Y 22.9340, Z -7.1667, A 0.000, B 0.000, C 0.000 }
gfCNCPoint5[25132] = {X 444.3942, Y 22.9560, Z -7.1667, A 0.000, B 0.000, C 0.000 }
gfCNCPoint5[25133] = {X 445.9305, Y 22.9560, Z -7.1667, A 0.000, B 0.000, C 0.000 }
gfCNCPoint5[25134] = {X 449.9305, Y 22.9560, Z -7.1667, A 0.000, B 0.000, C 0.000 }
gfCNCPoint5[25135] = {X 449.9305, Y 22.9560, Z -4.1667, A 0.000, B 0.000, C 0.000 }
gfCNCPoint5[25136] = {X 449.9305, Y 22.9560, Z 11.0000, A 0.000, B 0.000, C 0.000 }
gfCNCPoint5[25137] = {X 491.9940, Y 19.7825, Z 11.0000, A 0.000, B 0.000, C 0.000 }
gfCNCPoint5[25138] = {X 491.9940, Y 19.7825, Z -3.3333, A 0.000, B 0.000, C 0.000 }
gfCNCPoint5[25139] = {X 487.6645, Y 19.7821, Z -4.4934, A 0.000, B 0.000, C 0.000 }
gfCNCPoint5[25140] = {X 486.9696, Y 19.7868, Z -4.6796, A 0.000, B 0.000, C 0.000 }
gfCNCPoint5[25141] = {X 486.2691, Y 19.7850, Z -4.8673, A 0.000, B 0.000, C 0.000 }
gfCNCPoint5[25142] = {X 485.4748, Y 19.8903, Z -5.0820, A 0.000, B 0.000, C 0.000 }
gfCNCPoint5[25143] = {X 484.7990, Y 20.0747, Z -5.2697, A 0.000, B 0.000, C 0.000 }
gfCNCPoint5[25144] = {X 484.6644, Y 20.1115, Z -5.3071, A 0.000, B 0.000, C 0.000 }
gfCNCPoint5[25145] = {X 484.6312, Y 20.1429, Z -5.3193, A 0.000, B 0.000, C 0.000 }
gfCNCPoint5[25146] = {X 484.5869, Y 20.2752, Z -5.3567, A 0.000, B 0.000, C 0.000 }
gfCNCPoint5[25147] = {X 484.4395, Y 20.7162, Z -5.4813, A 0.000, B 0.000, C 0.000 }
gfCNCPoint5[25148] = {X 484.4054, Y 21.9049, Z -5.8000, A 0.000, B 0.000, C 0.000 }
gfCNCPoint5[25149] = {X 484.5273, Y 22.3535, Z -5.9245, A 0.000, B 0.000, C 0.000 }
gfCNCPoint5[25150] = {X 484.7222, Y 22.4168, Z -5.9794, A 0.000, B 0.000, C 0.000 }
gfCNCPoint5[25151] = {X 484.9347, Y 22.4345, Z -6.0366, A 0.000, B 0.000, C 0.000 }
gfCNCPoint5[25152] = {X 486.1028, Y 22.5563, Z -6.3513, A 0.000, B 0.000, C 0.000 }
gfCNCPoint5[25153] = {X 486.4648, Y 22.5726, Z -6.4484, A 0.000, B 0.000, C 0.000 }
gfCNCPoint5[25154] = {X 487.6448, Y 22.5560, Z -6.7646, A 0.000, B 0.000, C 0.000 }
gfCNCPoint5[25155] = {X 489.1455, Y 22.5560, Z -7.1667, A 0.000, B 0.000, C 0.000 }
gfCNCPoint5[25156] = {X 493.3690, Y 22.5560, Z -7.1667, A 0.000, B 0.000, C 0.000 }
gfCNCPoint5[25157] = {X 493.3690, Y 19.7826, Z -7.1667, A 0.000, B 0.000, C 0.000 }
gfCNCPoint5[25158] = {X 487.6645, Y 19.7821, Z -7.1667, A 0.000, B 0.000, C 0.000 }
gfCNCPoint5[25159] = {X 486.9696, Y 19.7868, Z -7.1667, A 0.000, B 0.000, C 0.000 }
gfCNCPoint5[25160] = {X 485.8746, Y 19.8577, Z -7.1667, A 0.000, B 0.000, C 0.000 }
gfCNCPoint5[25161] = {X 484.7990, Y 20.0747, Z -7.1667, A 0.000, B 0.000, C 0.000 }
gfCNCPoint5[25162] = {X 484.6679, Y 20.1484, Z -7.1667, A 0.000, B 0.000, C 0.000 }
gfCNCPoint5[25163] = {X 484.5869, Y 20.2752, Z -7.1667, A 0.000, B 0.000, C 0.000 }
gfCNCPoint5[25164] = {X 484.4306, Y 20.9596, Z -7.1667, A 0.000, B 0.000, C 0.000 }
gfCNCPoint5[25165] = {X 484.4104, Y 21.6613, Z -7.1667, A 0.000, B 0.000, C 0.000 }
gfCNCPoint5[25166] = {X 484.5273, Y 22.3535, Z -7.1667, A 0.000, B 0.000, C 0.000 }
gfCNCPoint5[25167] = {X 484.7286, Y 22.4061, Z -7.1667, A 0.000, B 0.000, C 0.000 }
gfCNCPoint5[25168] = {X 484.9347, Y 22.4345, Z -7.1667, A 0.000, B 0.000, C 0.000 }
gfCNCPoint5[25169] = {X 486.2879, Y 22.5353, Z -7.1667, A 0.000, B 0.000, C 0.000 }
gfCNCPoint5[25170] = {X 487.6448, Y 22.5560, Z -7.1667, A 0.000, B 0.000, C 0.000 }
gfCNCPoint5[25171] = {X 489.1455, Y 22.5560, Z -7.1667, A 0.000, B 0.000, C 0.000 }
gfCNCPoint5[25172] = {X 485.1607, Y 22.2874, Z -7.1667, A 0.000, B 0.000, C 0.000 }
gfCNCPoint5[25173] = {X 489.1455, Y 22.6360, Z -7.1667, A 0.000, B 0.000, C 0.000 }
gfCNCPoint5[25174] = {X 493.4490, Y 22.6360, Z -7.1667, A 0.000, B 0.000, C 0.000 }
gfCNCPoint5[25175] = {X 493.4490, Y 19.7026, Z -7.1667, A 0.000, B 0.000, C 0.000 }
gfCNCPoint5[25176] = {X 487.6642, Y 19.7021, Z -7.1667, A 0.000, B 0.000, C 0.000 }
gfCNCPoint5[25177] = {X 486.9713, Y 19.7068, Z -7.1667, A 0.000, B 0.000, C 0.000 }
gfCNCPoint5[25178] = {X 485.8649, Y 19.7783, Z -7.1667, A 0.000, B 0.000, C 0.000 }
gfCNCPoint5[25179] = {X 484.7780, Y 19.9975, Z -7.1667, A 0.000, B 0.000, C 0.000 }
gfCNCPoint5[25180] = {X 484.6129, Y 20.0903, Z -7.1667, A 0.000, B 0.000, C 0.000 }
gfCNCPoint5[25181] = {X 484.5111, Y 20.2498, Z -7.1667, A 0.000, B 0.000, C 0.000 }
gfCNCPoint5[25182] = {X 484.3494, Y 20.9636, Z -7.1667, A 0.000, B 0.000, C 0.000 }
gfCNCPoint5[25183] = {X 484.3327, Y 21.6953, Z -7.1667, A 0.000, B 0.000, C 0.000 }
gfCNCPoint5[25184] = {X 484.4616, Y 22.4158, Z -7.1667, A 0.000, B 0.000, C 0.000 }
gfCNCPoint5[25185] = {X 484.6887, Y 22.4795, Z -7.1667, A 0.000, B 0.000, C 0.000 }
gfCNCPoint5[25186] = {X 484.9221, Y 22.5137, Z -7.1667, A 0.000, B 0.000, C 0.000 }
gfCNCPoint5[25187] = {X 486.2805, Y 22.6151, Z -7.1667, A 0.000, B 0.000, C 0.000 }
gfCNCPoint5[25188] = {X 487.6425, Y 22.6360, Z -7.1667, A 0.000, B 0.000, C 0.000 }
